       IF #Sts_PosAxis = 2 AND NOT #Alarm.CheckBothAxMove THEN
               //
               #Ax_Testa.CIn.Manager.MoveToPos := #Ctrl.Ax.OP_MoveToPos AND #Sts.Op_MoveToPos_Cnd;
               #Ax_Coda.CIn.Manager.MoveToPos := #Ctrl.Ax.OP_MoveToPos AND #Sts.Op_MoveToPos_Cnd;
               #Ax_Testa.CIn.Manager.Pos := #Ax_Coda.CIn.Manager.Pos := #CIn.Manager.Pos;

       END_IF;


       // ##########################
   (*    
   IF #Ctrl.Ax.OP_MoveToPos AND #Sts.Op_MoveToPos_Cnd AND NOT #Ax_Testa.COut.InPosition AND #Sollevatore_Testa.COut.Rest
       AND ( NOT #Alarm.Testa.Ax.S120_Fault AND NOT #Alarm.Coda.Ax.S120_Fault) THEN
       #Ax_Testa.CIn.Manager.MoveToPos := TRUE;

       // Se raggiungo la posizione di setpoint spengo il comando
   ELSIF #Ax_Testa.COut.InPosition AND #Ax_Testa.COut.Standstill OR ( #Alarm.Testa.Ax.S120_Fault OR #Alarm.Coda.Ax.S120_Fault) THEN
       #Ax_Testa.CIn.Manager.MoveToPos := FALSE;
       #Ax_Testa.DSI.PowerEnable := FALSE;
   END_IF;

   // MANIPOLATORE CODA
   #Ax_Coda.CIn.Manager.Control_ON := #Ax_Coda.DSI.PowerEnable
   := #Sollevatore_Coda.Cin.Manager.Control_ON := #Magnete_Coda.Cin.Manager.Control_ON := #Ctrl.Ax.OP_MoveToPos;

   IF #Ctrl.Ax.OP_MoveToPos AND #Sts.Op_MoveToPos_Cnd AND NOT #Ax_Coda.COut.InPosition AND #Sollevatore_Coda.COut.Rest
       AND ( NOT #Alarm.Testa.Ax.S120_Fault AND NOT #Alarm.Coda.Ax.S120_Fault) THEN
           #Ax_Coda.CIn.Manager.MoveToPos := TRUE;

           // Se raggiungo la posizione di setpoint spengo il comando
       ELSIF #Ax_Coda.COut.InPosition AND #Ax_Coda.COut.Standstill OR ( #Alarm.Testa.Ax.S120_Fault OR #Alarm.Coda.Ax.S120_Fault) THEN
           #Ax_Coda.CIn.Manager.MoveToPos := FALSE;
           #Ax_Coda.DSI.PowerEnable := FALSE;
       END_IF;
       *)
END_REGION

REGION Network 55 (SCL): [Sollevamento] - Cin Manager (Esecuzione sequenza comandi)
   // Comando CIn Manager ControlON di tutte le utenze
   // MANIPOLATORE TESTA & CODA
   #Sollevatore_Testa.Cin.Manager.Control_ON := #CIn.Manager.Control_ON;
   #Sollevatore_Coda.Cin.Manager.Control_ON := #CIn.Manager.Control_ON;
   //
   #Sollevatore_Testa.Cin.Manager.Rest := FALSE;
   #Sollevatore_Testa.Cin.Manager.Work := FALSE;
   #Sollevatore_Coda.Cin.Manager.Rest := FALSE;
   #Sollevatore_Coda.Cin.Manager.Work := FALSE;

   // Gestione dei comandi relativi a Sollevamento in sequenza quando ho un OP cnd

   IF (#Ctrl.Sollevamento.OP_Rest AND #Sts.Sollevamento.OP_Rest_Cnd) THEN

       #Sollevatore_Testa.Cin.Manager.Rest := TRUE;
       #Sollevatore_Coda.Cin.Manager.Rest := TRUE;

           // Vado a lavoro solo se sono in posizione    
   ELSIF  (#Ctrl.Sollevamento.OP_Work AND #Sts.Sollevamento.Op_Work_Cnd) AND (#COut.InPos_Prelievo OR #COut.InPos_BancoScarto OR #COut.InPos_BancoA0303) THEN

       #Sollevatore_Testa.Cin.Manager.Work := TRUE;
       #Sollevatore_Coda.Cin.Manager.Work := TRUE;

   END_IF;
END_REGION

REGION Network 56 (SCL): [Magneti] - Cin Manager (Esecuzione sequenza comandi)


   // Comando CIn Manager ControlON di tutte le utenze
   // MAGNETI TESTA & CODA
   #Magnete_Testa.Cin.Manager.Control_ON := (#Ctrl.Magneti.OP_Rest OR #Ctrl.Magneti.OP_Work) OR (#Ctrl.Sollevamento.OP_Rest OR #Ctrl.Sollevamento.OP_Work);
   #Magnete_Coda.Cin.Manager.Control_ON := (#Ctrl.Magneti.OP_Rest OR #Ctrl.Magneti.OP_Work) OR (#Ctrl.Sollevamento.OP_Rest OR #Ctrl.Sollevamento.OP_Work);
   //
   // Gestione dei comandi relativi ai Magneti in sequenza quando ho un OP cnd
   IF (#Ctrl.Magneti.OP_Rest AND #Sts.Magneti.OP_Rest_Cnd) AND #Sollevatore_Testa.COut.Work AND #Sollevatore_Coda.COut.Work THEN

       #Magnete_Testa.Cin.Manager.Work := FALSE;
       #Magnete_Coda.Cin.Manager.Work := FALSE;
       #Magnete_Testa.Cin.Manager.Rest := TRUE;
       #Magnete_Coda.Cin.Manager.Rest := TRUE;

   ELSIF (#Ctrl.Magneti.OP_Rest AND #Sts.Magneti.OP_Rest_Cnd) AND #COut.InPos_BancoScarto THEN

       #Magnete_Testa.Cin.Manager.Work := FALSE;
       #Magnete_Coda.Cin.Manager.Work := FALSE;
       #Magnete_Testa.Cin.Manager.Rest := TRUE;
       #Magnete_Coda.Cin.Manager.Rest := TRUE;

           // Vado a lavoro solo se sono in posizione e il sollevatore è a lavoro    
   ELSIF  (#Ctrl.Magneti.OP_Work AND #Sts.Magneti.Op_Work_Cnd) THEN

       #Magnete_Testa.Cin.Manager.Rest := FALSE;
       #Magnete_Coda.Cin.Manager.Rest := FALSE;
       #Magnete_Testa.Cin.Manager.Work := TRUE;
       #Magnete_Coda.Cin.Manager.Work := TRUE;

   END_IF;
END_REGION

REGION Network 58: <<< MACHINE STATUS >>>
END_REGION

REGION Network 59: Collect machine to zone interface (internal machines OR)
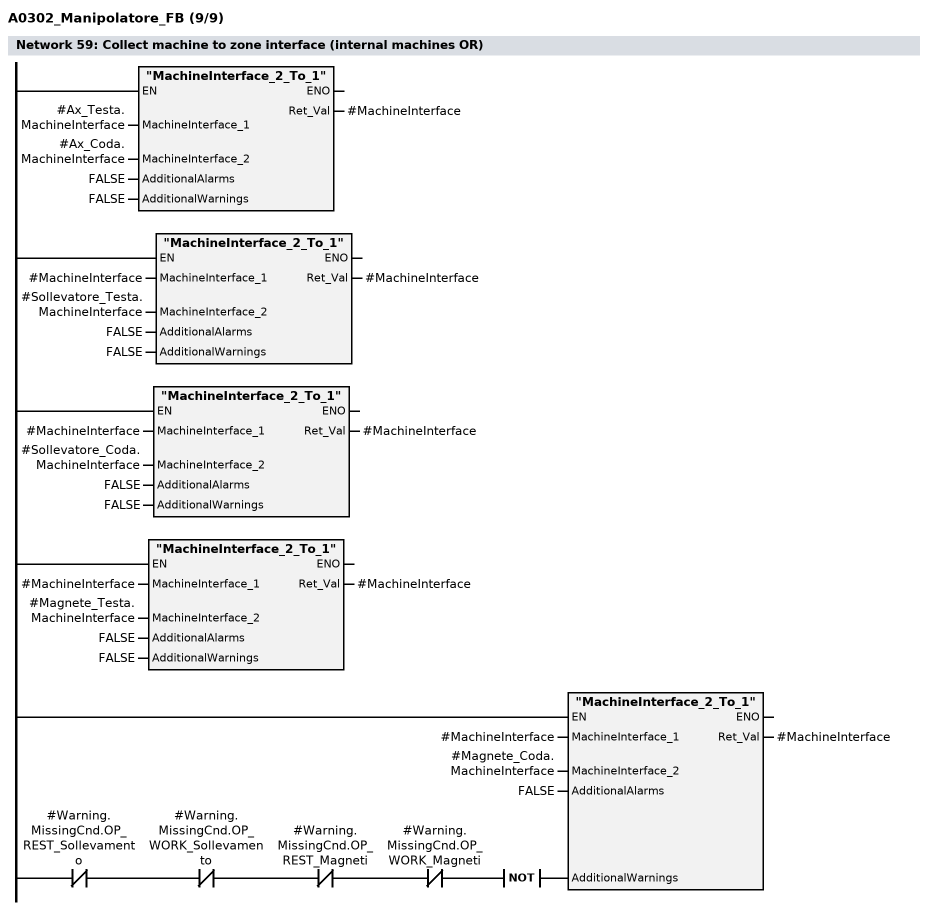
   RUNG wire#powerrail
      "MachineInterface_2_To_1"(MachineInterface_1 := #Ax_Testa.MachineInterface, MachineInterface_2 := #Ax_Coda.MachineInterface, AdditionalAlarms := FALSE, AdditionalWarnings := FALSE, Ret_Val => #MachineInterface)
   END_RUNG
   RUNG wire#powerrail
      "MachineInterface_2_To_1"(MachineInterface_1 := #MachineInterface, MachineInterface_2 := #Sollevatore_Testa.MachineInterface, AdditionalAlarms := FALSE, AdditionalWarnings := FALSE, Ret_Val => #MachineInterface)
   END_RUNG
   RUNG wire#powerrail
      "MachineInterface_2_To_1"(MachineInterface_1 := #MachineInterface, MachineInterface_2 := #Sollevatore_Coda.MachineInterface, AdditionalAlarms := FALSE, AdditionalWarnings := FALSE, Ret_Val => #MachineInterface)
   END_RUNG
   RUNG wire#powerrail
      "MachineInterface_2_To_1"(MachineInterface_1 := #MachineInterface, MachineInterface_2 := #Magnete_Testa.MachineInterface, AdditionalAlarms := FALSE, AdditionalWarnings := FALSE, Ret_Val => #MachineInterface)
   END_RUNG
   RUNG wire#powerrail
      "MachineInterface_2_To_1"(AdditionalWarnings := wire#w1, MachineInterface_1 := #MachineInterface, MachineInterface_2 := #Magnete_Coda.MachineInterface, AdditionalAlarms := FALSE, Ret_Val => #MachineInterface)
   END_RUNG
   RUNG wire#powerrail
      I_Contact( #Warning.MissingCnd.OP_REST_Sollevamento )
      I_Contact( #Warning.MissingCnd.OP_WORK_Sollevamento )
      I_Contact( #Warning.MissingCnd.OP_REST_Magneti )
      I_Contact( #Warning.MissingCnd.OP_WORK_Magneti )
      Not()
   END_RUNG wire#w1
   // the same network as SCL:
   #MachineInterface := "MachineInterface_2_To_1"(MachineInterface_1 := #Ax_Testa.MachineInterface,
                           MachineInterface_2 := #Ax_Coda.MachineInterface,
                           AdditionalAlarms := FALSE,
                           AdditionalWarnings := FALSE);
   #MachineInterface := "MachineInterface_2_To_1"(MachineInterface_1 := #MachineInterface,
                           MachineInterface_2 := #Sollevatore_Testa.MachineInterface,
                           AdditionalAlarms := FALSE,
                           AdditionalWarnings := FALSE);
   #MachineInterface := "MachineInterface_2_To_1"(MachineInterface_1 := #MachineInterface,
                           MachineInterface_2 := #Sollevatore_Coda.MachineInterface,
                           AdditionalAlarms := FALSE,
                           AdditionalWarnings := FALSE);
   #MachineInterface := "MachineInterface_2_To_1"(MachineInterface_1 := #MachineInterface,
                           MachineInterface_2 := #Magnete_Testa.MachineInterface,
                           AdditionalAlarms := FALSE,
                           AdditionalWarnings := FALSE);
   #MachineInterface := "MachineInterface_2_To_1"(MachineInterface_1 := #MachineInterface,
                           MachineInterface_2 := #Magnete_Coda.MachineInterface,
                           AdditionalAlarms := FALSE,
                           AdditionalWarnings := NOT (NOT #Warning.MissingCnd.OP_REST_Sollevamento AND NOT #Warning.MissingCnd.OP_WORK_Sollevamento AND NOT #Warning.MissingCnd.OP_REST_Magneti AND NOT #Warning.MissingCnd.OP_WORK_Magneti));
END_REGION
END_FUNCTION_BLOCK

FUNCTION "A0302_Bordatrice_RegolazioneFormato_OB1_CALL" : Void   // FC151, LAD
// stored: SetENOAutomatically false
   VAR_TEMP
      RETVAL_SET_CINT : Int;
      Check_Low : Bool;
      ChecK_High : Bool;
   END_VAR
   VAR_TEMP   // added for the SCL form of the ladder/FBD networks
      _w1 : Bool;
      _w2 : Bool;
      _w3 : Bool;
   END_VAR
BEGIN

REGION Network 2
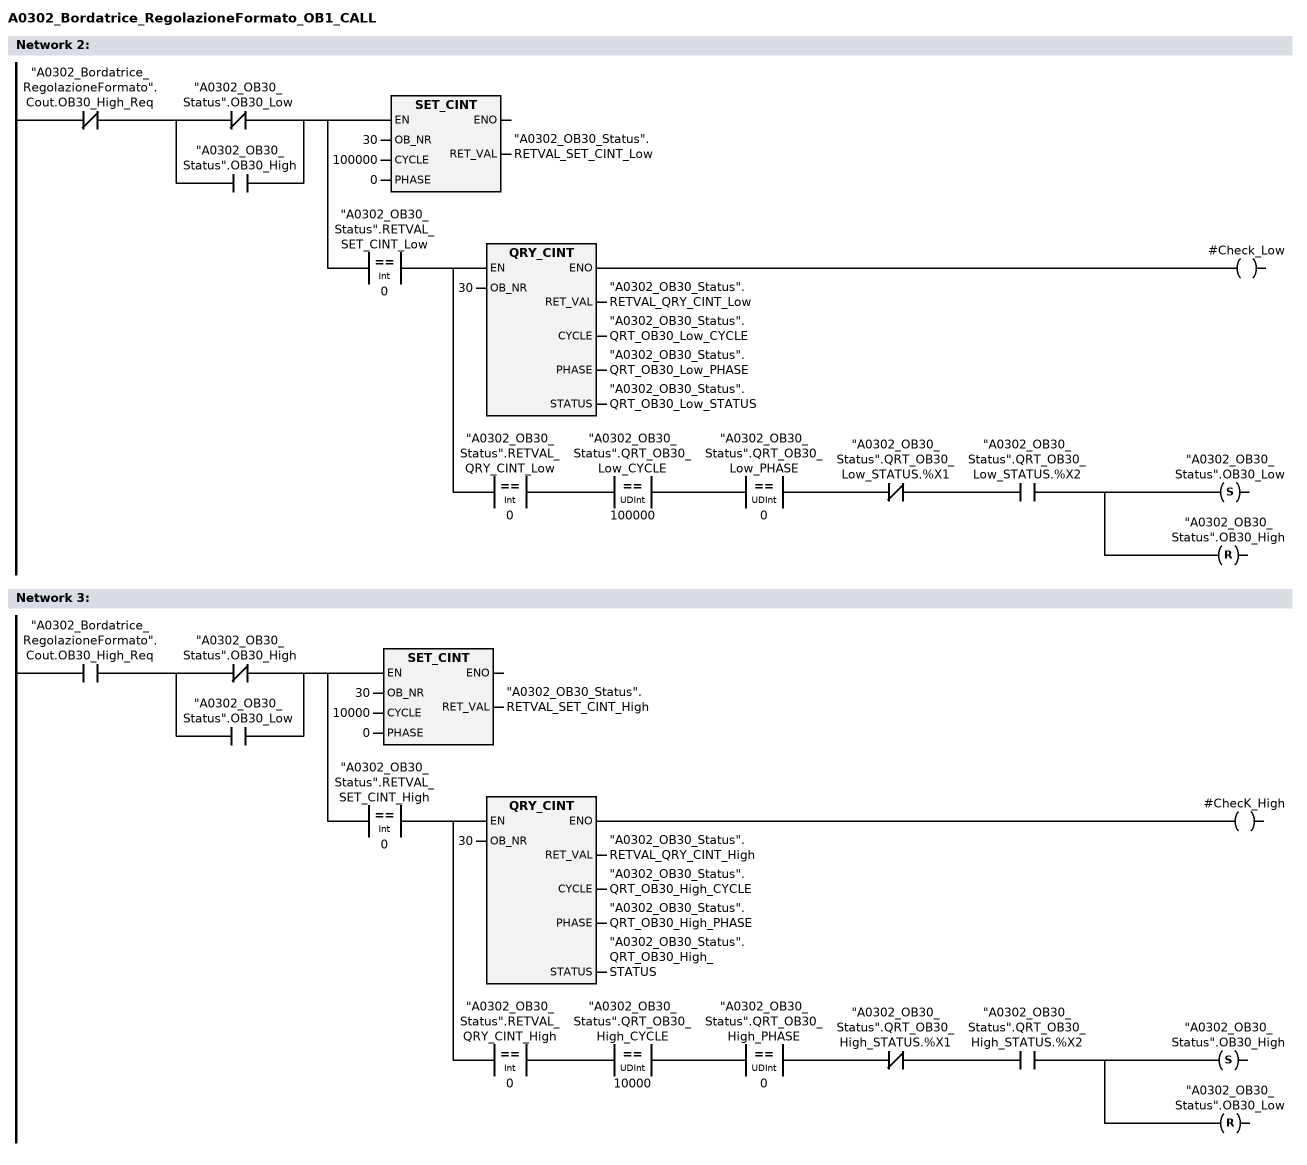
   RUNG wire#powerrail
      I_Contact( "A0302_Bordatrice_RegolazioneFormato".Cout.OB30_High_Req )
      wire#w1
      I_Contact( "A0302_OB30_Status".OB30_Low )
      wire#w2
      SET_CINT(OB_NR := 30, CYCLE := 100000, PHASE := 0, RET_VAL => "A0302_OB30_Status".RETVAL_SET_CINT_Low)
   END_RUNG
   RUNG wire#w1
      Contact( "A0302_OB30_Status".OB30_High )
   END_RUNG wire#w2
   RUNG wire#w2
      { S7_Templates := "SrcType := Int" } EQ_Contact(in1 := "A0302_OB30_Status".RETVAL_SET_CINT_Low, in2 := 0)
      wire#w3
      QRY_CINT(OB_NR := 30, RET_VAL => "A0302_OB30_Status".RETVAL_QRY_CINT_Low, CYCLE => "A0302_OB30_Status".QRT_OB30_Low_CYCLE, PHASE => "A0302_OB30_Status".QRT_OB30_Low_PHASE, STATUS => "A0302_OB30_Status".QRT_OB30_Low_STATUS)
      Coil( #Check_Low )
   END_RUNG
   RUNG wire#w3
      { S7_Templates := "SrcType := Int" } EQ_Contact(in1 := "A0302_OB30_Status".RETVAL_QRY_CINT_Low, in2 := 0)
      { S7_Templates := "SrcType := UDInt" } EQ_Contact(in1 := "A0302_OB30_Status".QRT_OB30_Low_CYCLE, in2 := 100000)
      { S7_Templates := "SrcType := UDInt" } EQ_Contact(in1 := "A0302_OB30_Status".QRT_OB30_Low_PHASE, in2 := 0)
      I_Contact( "A0302_OB30_Status".QRT_OB30_Low_STATUS.%X1 )
      Contact( "A0302_OB30_Status".QRT_OB30_Low_STATUS.%X2 )
      wire#w4
      S_Coil( "A0302_OB30_Status".OB30_Low )
   END_RUNG
   RUNG wire#w4
      R_Coil( "A0302_OB30_Status".OB30_High )
   END_RUNG
   // the same network as SCL:
   #_w1 := NOT "A0302_Bordatrice_RegolazioneFormato".Cout.OB30_High_Req AND (NOT "A0302_OB30_Status".OB30_Low OR "A0302_OB30_Status".OB30_High);
   IF #_w1 THEN
       "A0302_OB30_Status".RETVAL_SET_CINT_Low := SET_CINT(OB_NR := 30, CYCLE := 100000, PHASE := 0);
   END_IF;
   #_w2 := #_w1 AND ("A0302_OB30_Status".RETVAL_SET_CINT_Low = 0);
   "A0302_OB30_Status".RETVAL_QRY_CINT_Low := QRY_CINT(EN := #_w2,
                           OB_NR := 30,
                           CYCLE => "A0302_OB30_Status".QRT_OB30_Low_CYCLE,
                           PHASE => "A0302_OB30_Status".QRT_OB30_Low_PHASE,
                           STATUS => "A0302_OB30_Status".QRT_OB30_Low_STATUS,
                           ENO => #_w3);
   #Check_Low := #_w3;
   IF #_w2 AND ("A0302_OB30_Status".RETVAL_QRY_CINT_Low = 0) AND ("A0302_OB30_Status".QRT_OB30_Low_CYCLE = 100000) AND ("A0302_OB30_Status".QRT_OB30_Low_PHASE = 0) AND NOT "A0302_OB30_Status".QRT_OB30_Low_STATUS.%X1 AND "A0302_OB30_Status".QRT_OB30_Low_STATUS.%X2 THEN
       "A0302_OB30_Status".OB30_Low := TRUE;
       "A0302_OB30_Status".OB30_High := FALSE;
   END_IF;
END_REGION

REGION Network 3
   RUNG wire#powerrail
      Contact( "A0302_Bordatrice_RegolazioneFormato".Cout.OB30_High_Req )
      wire#w1
      I_Contact( "A0302_OB30_Status".OB30_High )
      wire#w2
      SET_CINT(OB_NR := 30, CYCLE := 10000, PHASE := 0, RET_VAL => "A0302_OB30_Status".RETVAL_SET_CINT_High)
   END_RUNG
   RUNG wire#w1
      Contact( "A0302_OB30_Status".OB30_Low )
   END_RUNG wire#w2
   RUNG wire#w2
      { S7_Templates := "SrcType := Int" } EQ_Contact(in1 := "A0302_OB30_Status".RETVAL_SET_CINT_High, in2 := 0)
      wire#w3
      QRY_CINT(OB_NR := 30, RET_VAL => "A0302_OB30_Status".RETVAL_QRY_CINT_High, CYCLE => "A0302_OB30_Status".QRT_OB30_High_CYCLE, PHASE => "A0302_OB30_Status".QRT_OB30_High_PHASE, STATUS => "A0302_OB30_Status".QRT_OB30_High_STATUS)
      Coil( #ChecK_High )
   END_RUNG
   RUNG wire#w3
      { S7_Templates := "SrcType := Int" } EQ_Contact(in1 := "A0302_OB30_Status".RETVAL_QRY_CINT_High, in2 := 0)
      { S7_Templates := "SrcType := UDInt" } EQ_Contact(in1 := "A0302_OB30_Status".QRT_OB30_High_CYCLE, in2 := 10000)
      { S7_Templates := "SrcType := UDInt" } EQ_Contact(in1 := "A0302_OB30_Status".QRT_OB30_High_PHASE, in2 := 0)
      I_Contact( "A0302_OB30_Status".QRT_OB30_High_STATUS.%X1 )
      Contact( "A0302_OB30_Status".QRT_OB30_High_STATUS.%X2 )
      wire#w4
      S_Coil( "A0302_OB30_Status".OB30_High )
   END_RUNG
   RUNG wire#w4
      R_Coil( "A0302_OB30_Status".OB30_Low )
   END_RUNG
   // the same network as SCL:
   #_w1 := "A0302_Bordatrice_RegolazioneFormato".Cout.OB30_High_Req AND (NOT "A0302_OB30_Status".OB30_High OR "A0302_OB30_Status".OB30_Low);
   IF #_w1 THEN
       "A0302_OB30_Status".RETVAL_SET_CINT_High := SET_CINT(OB_NR := 30, CYCLE := 10000, PHASE := 0);
   END_IF;
   #_w2 := #_w1 AND ("A0302_OB30_Status".RETVAL_SET_CINT_High = 0);
   "A0302_OB30_Status".RETVAL_QRY_CINT_High := QRY_CINT(EN := #_w2,
                           OB_NR := 30,
                           CYCLE => "A0302_OB30_Status".QRT_OB30_High_CYCLE,
                           PHASE => "A0302_OB30_Status".QRT_OB30_High_PHASE,
                           STATUS => "A0302_OB30_Status".QRT_OB30_High_STATUS,
                           ENO => #_w3);
   #ChecK_High := #_w3;
   IF #_w2 AND ("A0302_OB30_Status".RETVAL_QRY_CINT_High = 0) AND ("A0302_OB30_Status".QRT_OB30_High_CYCLE = 10000) AND ("A0302_OB30_Status".QRT_OB30_High_PHASE = 0) AND NOT "A0302_OB30_Status".QRT_OB30_High_STATUS.%X1 AND "A0302_OB30_Status".QRT_OB30_High_STATUS.%X2 THEN
       "A0302_OB30_Status".OB30_High := TRUE;
       "A0302_OB30_Status".OB30_Low := FALSE;
   END_IF;
END_REGION
END_FUNCTION

FUNCTION "A0302_Bordatrice_CALL" : Void   // FC181, LAD
TITLE = << BORDATRICE MOVIMENTO >>
// stored: SetENOAutomatically false
   VAR CONSTANT
      MinimumPos : Real := 0.0;
      MaximumPos : Real := 1000.0;
      MISSING : Int;
   END_VAR
BEGIN

REGION Network 1 (SCL): << TRASFERIMENTO stati CIn del blocco >>
   // SOSTITUIRE SYS BYPASS CON INGRESSI DIGITALI

   // TRASFERIMENTO COMANDI CIn MANAGER
   "A0302_Bordatrice".CIn.Manager.Ax := "A0302_Manager".COut.Bordatrice.Ax;
   //
   "A0302_Bordatrice".CIn.SemiAut_Pb := "A0302_Manager".DataIn.SemiAut_Pb;


   REGION TRASFERIMENTO CIn DIGITAL INPUT dei LIMIT SWITCH
       //
       //"A0302_Bordatrice".Ax.CIn.PositionLimits.EnableMin := FALSE;
       //"A0302_Bordatrice".Ax.CIn.PositionLimits.EnableMax := FALSE;

   END_REGION ;

   REGION TRASFERIMENTO STATI STAZIONE P5

       "A0302_Bordatrice".CIn.P5.Sollevatori := "A0301_Spintore_Lat".COut.Sollevatori;
       "A0302_Bordatrice".CIn.P5.SpintoreLong := "A0302_Spintore".COut.Spintore;
       "A0302_Bordatrice".CIn.P5.Sens.FTC_Ingombro_A0301 := "A0302_Spintore".IEC.FTC_On;

   END_REGION ;

   REGION  TRASFERIMENTO STATI RULLIERA dopo BORDATRICE

       "A0302_Bordatrice".CIn.Rulliera.Centratori := "A0302_Centratori".COut.Centraggio;
       "A0302_Bordatrice".CIn.Rulliera.Sollevatori := "A0302_Centratori".COut.Sollevamento;
       "A0302_Bordatrice".CIn.Rulliera.Coda.Sens := "A0302_Manager".CIn.Rulliera.Coda.Sens;
       "A0302_Bordatrice".CIn.Rulliera.Centro.Sens := "A0302_Manager".CIn.Rulliera.Centro.Sens;

   END_REGION ;

   REGION TRASFERIMENTO STATI CARRO PAREGGIATORE DI CODA

       "A0302_Bordatrice".CIn.CarroPareggCoda.Ax := "A0302_PareggiatoreCoda".COut.Ax;
       "A0302_Bordatrice".CIn.CarroPareggCoda.Bloccaggio := "A0302_PareggiatoreCoda".COut.Bloccaggio;
       "A0302_Bordatrice".CIn.CarroPareggCoda.BattutaVerticale := "A0302_PareggiatoreCoda".COut.BattutaVerticale;
       "A0302_Bordatrice".CIn.CarroPareggCoda.PareggiatoreLongitudinale := "A0302_PareggiatoreCoda".COut.PareggiatoreLong;
       "A0302_Bordatrice".CIn.CarroPareggCoda.Sens := "A0302_Manager".CIn.CarroPareggCoda.Sens;

   END_REGION ;

   REGION  TRASFERIMENTO STATI CARRO PAREGGIATORE DI TESTA

       "A0302_Bordatrice".CIn.CarroPareggTesta.Ax := "A0302_PareggiatoreTesta".COut.Ax;
       "A0302_Bordatrice".CIn.CarroPareggTesta.Bloccaggio := "A0302_PareggiatoreTesta".COut.Bloccaggio;
       "A0302_Bordatrice".CIn.CarroPareggTesta.Centraggio := "A0302_PareggiatoreTesta".COut.Centraggio;
       "A0302_Bordatrice".CIn.CarroPareggTesta.Sollevatore := "A0302_PareggiatoreTesta".COut.Sollevatore;
       "A0302_Bordatrice".CIn.CarroPareggTesta.Sens := "A0302_Manager".CIn.CarroPareggTesta.Sens;

   END_REGION ;

   // ATTREZZAGGIO PRONTO
   "A0302_Bordatrice".CIn.Attrezzaggio.CarriParegg.Ready := "A0302_Manager".Sts.Attrezzamento.Ready;
END_REGION

REGION Network 2 (SCL): << TRASFERIMENTO stati DataIn >>
   REGION TRASFERIMENTO #DataIn STATI BUTTON BORDATRICE
       // PB BORDATRICE
       "A0302_Bordatrice".Ax.DataIn.PB.Bwd_Minus := "A03_HMI".MB3.Button.A0302.Bordatrice.Ax.Bwd_Minus;
       "A0302_Bordatrice".Ax.DataIn.PB.Fwd_Plus := "A03_HMI".MB3.Button.A0302.Bordatrice.Ax.Fwd_Plus;
       "A0302_Bordatrice".Ax.DataIn.PB.MoveToPos := "A03_HMI".MB3.Button.A0302.Bordatrice.Ax.MoveToPos;

       // Sensori
       "A0302_Bordatrice".DataIn.Sens.FTC_Uscita := "A0302_Bordatrice_Banco_4_Lato_1_Phc_AtExit";

       // Feedback connettori
       "A0302_Bordatrice".DataIn.FdBack.ConnMotori := "A0302_Bordatrice_ControlloConnettoreBanco_4_Lato_1";
       "A0302_Bordatrice".DataIn.FdBack.ConnAux := "A0302_Bordatrice_ControlloConnettoreBanco_4_Lato_2";

   END_REGION ;
END_REGION

REGION Network 3 (SCL): DSI
   //
   "A0302_Bordatrice".DSI := "F_DB".DSI_S120_Bordatrice;
END_REGION

REGION Network 4 (SCL): HW
   //
   "A0302_Bordatrice".HWID_TEL111 := "HW_Const_Values".CU5_PN_1950A1_SIEMENS_telegram_111;
END_REGION

REGION Network 5 (SCL): Drive
   //
   "A0302_Bordatrice".Drive.Infeed_ON := "Areas_ITF".AG.Infeed_Running;
   "A0302_Bordatrice".Drive.AccessPoint := "HW_Const_Values".CU5_PN_1950A1_ModuleAccessPoint;
   "A0302_Bordatrice".Drive.AxisID := "CU5_ID_2_1950A1_1950M1";
   "A0302_Bordatrice".Drive.TokenChain := "TOKENCHAIN_CU5";
END_REGION

REGION Network 6: [Bordatrice] - Machine call
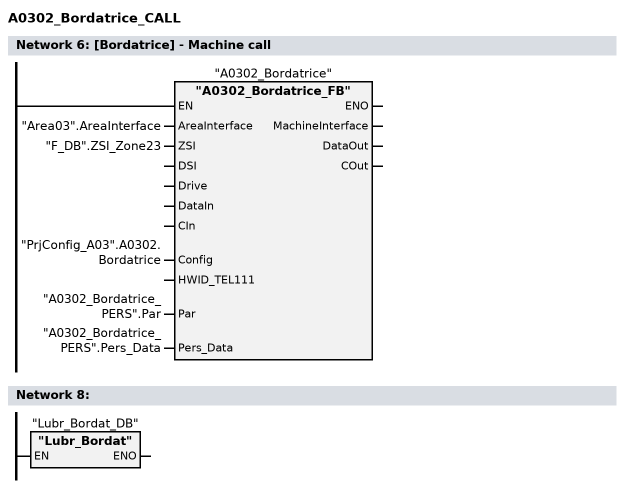
   RUNG wire#powerrail
      "A0302_Bordatrice"(AreaInterface := "Area03".AreaInterface, ZSI := "F_DB".ZSI_Zone23, DSI :=, Drive :=, DataIn :=, CIn :=, Config := "PrjConfig_A03".A0302.Bordatrice, HWID_TEL111 :=, Par := "A0302_Bordatrice_PERS".Par, Pers_Data := "A0302_Bordatrice_PERS".Pers_Data, MachineInterface =>, DataOut =>, COut =>)
   END_RUNG
   // the same network as SCL:
   "A0302_Bordatrice"(AreaInterface := "Area03".AreaInterface,   // "A0302_Bordatrice_FB"
                      ZSI := "F_DB".ZSI_Zone23,
                      Config := "PrjConfig_A03".A0302.Bordatrice,
                      Par := "A0302_Bordatrice_PERS".Par,
                      Pers_Data := "A0302_Bordatrice_PERS".Pers_Data);
END_REGION

REGION Network 8
   RUNG wire#powerrail
      "Lubr_Bordat_DB"()
   END_RUNG
   // the same network as SCL:
   "Lubr_Bordat_DB"();   // "Lubr_Bordat"
END_REGION
END_FUNCTION

FUNCTION_BLOCK "A0302_Bordatrice_FB"   // FB2, LAD
TITLE = == GESTIONE DELLA STAZIONE BORDATRICE ==
// stored: MemoryReserve 100, SetENOAutomatically false
   VAR_INPUT
      AreaInterface : "AreaInterface";
      ZSI : "udt_ZoneSafetyInterface";
      DSI : "udt_DeviceSafetyInterface";
      Drive : "TAx_DriveInterface";
      DataIn : Struct
         OP : "Ax_PB";
         Sens { ExternalAccessible := 'False'; ExternalVisible := 'False'; ExternalWritable := 'False'} : Struct
            FTC_Uscita : Bool;
         END_STRUCT;
         FdBack : Struct
            ConnMotori : Bool;
            ConnAux : Bool;
         END_STRUCT;
      END_STRUCT;
      CIn { ExternalAccessible := 'False'; ExternalVisible := 'False'; ExternalWritable := 'False'} : Struct
         Manager : Struct
            Ax : "Positioning_EPOS_Machine_Manager";
            Ax_Req : Struct
               Pos0 : Bool;
               Pos1 : Bool;
               Pos2 : Bool;
               Pos3 : Bool;
            END_STRUCT;
         END_STRUCT;
         SemiAut_Pb : Bool;
         P5 : Struct
            Sollevatori : "ValveMachine_COut";
            SpintoreLong : "ValveMachine_COut";
            Sens : Struct
               FTC_Ingombro_A0301 : Bool;   // 1614BF1 - I50.7
            END_STRUCT;
         END_STRUCT;
         Rulliera : Struct
            Ax_1 : "SpeedMachine_COut";
            Centratori : "ValveMachine_COut";
            Sollevatori : "ValveMachine_COut";
            Coda : Struct
               Sens : Struct
                  FTC_Rall : Bool;   // Sensori presenza materiale banco rallentamento ingresso
                  FTC_Prox_Ing : Bool;   // Sensori presenza materiale banco limite ingresso
               END_STRUCT;
            END_STRUCT;
            Centro : Struct
               Sens : Struct
                  FTC_Centrale : Bool;   // 2010BF1 - I50.2
               END_STRUCT;
            END_STRUCT;
         END_STRUCT;
         CarroPareggCoda : Struct
            Ax : "Positioning_DOL_Machine_COut";
            Bloccaggio : "ValveMachine_COut";
            BattutaVerticale : "ValveMachine_COut";
            PareggiatoreLongitudinale : "ValveMachine_COut";
            Sens : Struct
               FTC_Ingombro_In : Bool;   // 2012BF1 - I50.0
               FTC_Ingombro_Out : Bool;   // 2012BF2 - I50.1
               PresenzaMat : Bool;   // FC presenza materiale agganciato lato paregg coda
               PosPareggLong : Struct
                  Value : LReal;
                  CheckMeasure : Bool;
                  Standstill : Bool;
               END_STRUCT;
            END_STRUCT;
         END_STRUCT;
         CarroPareggTesta : Struct
            Ax : "Positioning_DOL_Machine_COut";
            Bloccaggio : "ValveMachine_COut";
            Centraggio : "ValveMachine_COut";
            Sollevatore : "ValveMachine_COut";
            Sens : Struct
               FTC1_Rall : Bool;   // 2010BF2 - I50.3
               FTC2_Prox_Ls : Bool;   // 2010BF3 - I50.4
               PresenzaMat : Bool;   // FC presenza materiale agganciato lato paregg testa
            END_STRUCT;
         END_STRUCT;
         Attrezzaggio : Struct
            CarriParegg : Struct
               Ready : Bool;
            END_STRUCT;
            BordRegFormato : Struct
               Ready : Bool;
            END_STRUCT;
         END_STRUCT;
      END_STRUCT;
      Config : Struct
         Ax : "Positioning_EPOS_Machine_Config_NEW";
         Measure : Struct
            K1_CarroPost : LReal;   // K1: Misura tra carro di coda e sensore applicato per controllo ingombro pezzo con carro giù
            K2_BancoIngresso : LReal;   // K2: Misura interasse tra lo 0 al centro del banco e la FTC all'uscita della Bordatrice
         END_STRUCT;
      END_STRUCT;
      HWID_TEL111 : HW_SUBMODULE;
   END_VAR
   VAR_OUTPUT
      MachineInterface { ExternalAccessible := 'False'; ExternalVisible := 'False'; ExternalWritable := 'False'} : "MachineInterface";
      DataOut : "Positioning_EPOS_Machine_DataOut";
      COut : Struct
         Ax : "Positioning_EPOS_Machine_COut";
         Ax_VelOveride : Struct
            Enable : Bool;
            Value : Real;
         END_STRUCT;
         Sts : Struct
            PosTargetEnable : Bool;
            PosTarget_Reached : Bool;
            In_W_Pos : Bool;
            AtRest : Bool;
         END_STRUCT;
         DataOut : "Positioning_EPOS_Machine_DataOut";
      END_STRUCT;
   END_VAR
   VAR_IN_OUT
      Par : Struct
         Ax_Man : "Positioning_EPOS_Machine_Par";
         Ax_Aut : "A0301_Mach_Speed_Par";
      END_STRUCT;
      Pers_Data : Struct
         EncoderAbsolute_Preset_OK : Bool;
         Persistent_ActualPosition : LReal;
      END_STRUCT;
   END_VAR
   VAR
      Alarm : Struct
         Ax { ExternalVisible := 'False'} : "Positioning_EPOS_Machine_Alr";
         StopIngombroCarroCoda : Bool;
         ConnMotori_FdBack : Bool;
         ConnAux_FdBack : Bool;
      END_STRUCT;
      Warning : Struct
         Ax { S7_SetPoint := 'True'} : "Positioning_EPOS_Machine_Wng";
         OP_REST_MissingCnd : Bool;   // Mancanza comando arresto
         OP_WORK_MissingCnd : Bool;   // Mancanza consenso lavoro
      END_STRUCT;
      Ax { S7_SetPoint := 'True'} : "Positioning_EPOS_Machine_FB_NEW";
      ValueVelOvr { ExternalAccessible := 'False'; ExternalVisible := 'False'; ExternalWritable := 'False'} : Array[1..10] of Real;
      Sts : Struct
         ReadyForMove : Bool;   // Pronto al movimento
         OP_CanMoveFreely : Bool;
         OP_MoveToPos_Cnd : Bool;
         OP_Bwd_Cnd : Bool;
         OP_Fwd_Cnd : Bool;
         Pz_UscitaBord : Bool;   // Pezzo in uscita dalla Bordatrice
         StopBordatrice : Bool;   // Stop Bordatrice da controllo quota spazio rimanente su rulliera di coda
         StandbyBordatrice : Bool;
      END_STRUCT;
      Ctrl : Struct
         Bordatrice : Struct
            OP_Bwd_Man : Bool;
            OP_Fwd_Man : Bool;
            OP_Bwd_Aut : Bool;
            OP_Fwd_Aut : Bool;
            OP_Bwd_Run : Bool;
            OP_Fwd_Run : Bool;
            OP_MoveToPos : Bool;
         END_STRUCT;
         Value : Struct
            Ax_TargetLongPos { ExternalAccessible := 'False'; ExternalVisible := 'False'; ExternalWritable := 'False'} : LReal;
            QuotaInizioUscita : LReal;
            QuotaFineUscita : LReal;
            PosTarget : LReal;
            QuotaRimanenteRullieraCoda : LReal;
         END_STRUCT;
         PosTargetEnable : Bool;
      END_STRUCT;
      HMI : Struct
         Pos : LReal;
      END_STRUCT;
      AUX : Struct
         Bordatrice : Struct
            OP_Bwd_Minus_PB : Bool;
            OP_Fwd_Plus_PB : Bool;
            OP_MoveToPos_PB { ExternalAccessible := 'False'; ExternalVisible := 'False'; ExternalWritable := 'False'} : Bool;
         END_STRUCT;
         Measure : Struct
            QuotaInizio : Bool;
            QuotaFine : Bool;
         END_STRUCT;
      END_STRUCT;
      IEC_FTC_UscitaBordatrice : Struct
         TON_Delay : IEC_TIMER;
         TOF_Delay { S7_SetPoint := 'True'} : IEC_TIMER;
         FTC_On { S7_SetPoint := 'True'} : Bool;
      END_STRUCT;
      IEC_StandbyBordatrice : IEC_TIMER;
      BTrk_Item : Struct
         BLean : Real;
         O_ID : DInt;
      END_STRUCT;
   END_VAR
   VAR_TEMP
      PE : Struct
         Bordatrice : Struct
            OP_Bwd_Minus_PB : Bool;
            OP_Fwd_Plus_PB : Bool;
            OP_MoveToPos_PB : Bool;
         END_STRUCT;
      END_STRUCT;
      VelOvr_Max : Real;   // Velocità max trovata
      i : Int;
      j : Int;
      CostB : LReal;
      Module : LReal;
      M_PosAPlusCostB : LReal;
      BTrk_GetData : Struct
         indx : Int;   // Se trovato tra i TODO / ENDING / OUT questo è l'indice dove sono stati prelevati i dati
         Sts : Int;   // 0 = Non Trovato; 0 = ACT; 1 = TODO; 2=ENDING; 3 = OUT
         Item : "Prod_Item_small";
      END_STRUCT;
      PositioningStop : Bool;
      NoTrk_Bordatrice : Bool;
   END_VAR
   VAR_TEMP   // added for the SCL form of the ladder/FBD networks
      _w1 : Bool;
      _w2 : Bool;
      _w3 : Bool;
      _w4 : Bool;
      _w5 : Bool;
      _w6 : Bool;
   END_VAR
BEGIN

REGION Network 1 (SCL): Reset allarmi
   IF #AreaInterface.RstAlarms THEN
       #Alarm.StopIngombroCarroCoda := FALSE;

       IF #DataIn.FdBack.ConnMotori AND #Alarm.ConnMotori_FdBack THEN
           #Alarm.ConnMotori_FdBack := FALSE;
       END_IF;

       IF #DataIn.FdBack.ConnAux AND #Alarm.ConnAux_FdBack THEN
           #Alarm.ConnAux_FdBack := FALSE;
       END_IF;
   END_IF;
   //
END_REGION

REGION Network 2: Controllo FdBack connettori
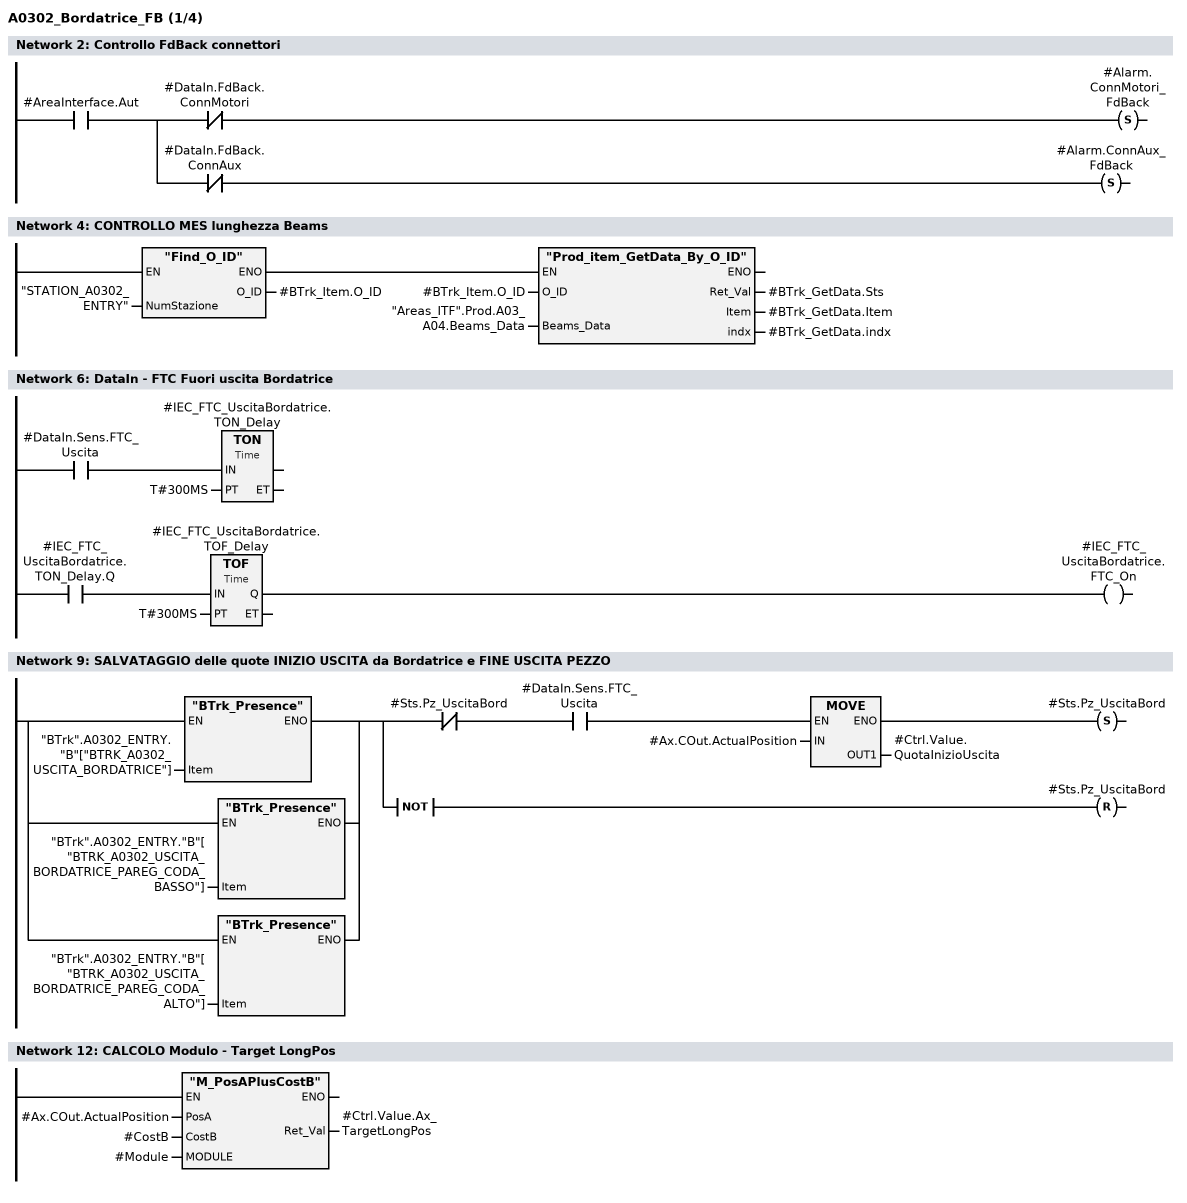
   RUNG wire#powerrail
      Contact( #AreaInterface.Aut )
      wire#w1
      I_Contact( #DataIn.FdBack.ConnMotori )
      S_Coil( #Alarm.ConnMotori_FdBack )
   END_RUNG
   RUNG wire#w1
      I_Contact( #DataIn.FdBack.ConnAux )
      S_Coil( #Alarm.ConnAux_FdBack )
   END_RUNG
   // the same network as SCL:
   IF #AreaInterface.Aut AND NOT #DataIn.FdBack.ConnMotori THEN #Alarm.ConnMotori_FdBack := TRUE; END_IF;
   IF #AreaInterface.Aut AND NOT #DataIn.FdBack.ConnAux THEN #Alarm.ConnAux_FdBack := TRUE; END_IF;
END_REGION

REGION Network 3: <+>
END_REGION

REGION Network 4: CONTROLLO MES lunghezza Beams
   RUNG wire#powerrail
      "Find_O_ID"(NumStazione := "STATION_A0302_ENTRY", O_ID => #BTrk_Item.O_ID)
      "Prod_item_GetData_By_O_ID"(O_ID := #BTrk_Item.O_ID, Beams_Data := "Areas_ITF".Prod.A03_A04.Beams_Data, Ret_Val => #BTrk_GetData.Sts, Item => #BTrk_GetData.Item, indx => #BTrk_GetData.indx)
   END_RUNG
   // the same network as SCL:
   "Find_O_ID"(NumStazione := "STATION_A0302_ENTRY", O_ID => #BTrk_Item.O_ID, ENO => #_w1);
   IF #_w1 THEN
       #BTrk_GetData.Sts := "Prod_item_GetData_By_O_ID"(O_ID := #BTrk_Item.O_ID,
                               Beams_Data := "Areas_ITF".Prod.A03_A04.Beams_Data,
                               Item => #BTrk_GetData.Item,
                               indx => #BTrk_GetData.indx);
   END_IF;
END_REGION

REGION Network 5 (SCL): CONTROLLO TRK lunghezza Beams
   //
   FOR #j:= 1 TO "BTRK_A0302_ENTRY_ITEMS" DO
       // 
       IF "BTrk".A0302_ENTRY.B[#j].BLen_Meas <> 0 THEN
           #BTrk_Item.BLean := "BTrk".A0302_ENTRY.B[#j].BLen_Meas;
       END_IF;

   END_FOR;
END_REGION

REGION Network 6: DataIn - FTC Fuori uscita Bordatrice
   RUNG wire#powerrail
      Contact( #DataIn.Sens.FTC_Uscita )
      { S7_Templates := "time_type := Time" } #IEC_FTC_UscitaBordatrice.TON_Delay.TON(pt := T#300MS, et =>)
   END_RUNG
   RUNG wire#powerrail
      Contact( #IEC_FTC_UscitaBordatrice.TON_Delay.Q )
      { S7_Templates := "time_type := Time" } #IEC_FTC_UscitaBordatrice.TOF_Delay.TOF(pt := T#300MS, et =>)
      Coil( #IEC_FTC_UscitaBordatrice.FTC_On )
   END_RUNG
   // the same network as SCL:
   #IEC_FTC_UscitaBordatrice.TON_Delay.TON(IN := #DataIn.Sens.FTC_Uscita, PT := T#300MS);
   #IEC_FTC_UscitaBordatrice.TOF_Delay.TOF(IN := #IEC_FTC_UscitaBordatrice.TON_Delay.Q, PT := T#300MS);
   #IEC_FTC_UscitaBordatrice.FTC_On := #IEC_FTC_UscitaBordatrice.TOF_Delay.Q;
END_REGION

REGION Network 7: <<<< CALCOLI QUOTE >>>>
END_REGION

REGION Network 8: <+>
END_REGION

REGION Network 9: SALVATAGGIO delle quote INIZIO USCITA da Bordatrice e FINE USCITA PEZZO
   RUNG wire#powerrail
      "BTrk_Presence"(Item := "BTrk".A0302_ENTRY."B"["BTRK_A0302_USCITA_BORDATRICE"])
      wire#w1
      I_Contact( #Sts.Pz_UscitaBord )
      Contact( #DataIn.Sens.FTC_Uscita )
      Move(in := #Ax.COut.ActualPosition, out1 => #Ctrl.Value.QuotaInizioUscita)
      S_Coil( #Sts.Pz_UscitaBord )
   END_RUNG
   RUNG wire#powerrail
      "BTrk_Presence"(Item := "BTrk".A0302_ENTRY."B"["BTRK_A0302_USCITA_BORDATRICE_PAREG_CODA_BASSO"])
   END_RUNG wire#w1
   RUNG wire#powerrail
      "BTrk_Presence"(Item := "BTrk".A0302_ENTRY."B"["BTRK_A0302_USCITA_BORDATRICE_PAREG_CODA_ALTO"])
   END_RUNG wire#w1
   RUNG wire#w1
      Not()
      R_Coil( #Sts.Pz_UscitaBord )
   END_RUNG
   // the same network as SCL:
   "BTrk_Presence"(Item := "BTrk".A0302_ENTRY."B"["BTRK_A0302_USCITA_BORDATRICE"], ENO => #_w1);
   "BTrk_Presence"(Item := "BTrk".A0302_ENTRY."B"["BTRK_A0302_USCITA_BORDATRICE_PAREG_CODA_BASSO"], ENO => #_w2);
   "BTrk_Presence"(Item := "BTrk".A0302_ENTRY."B"["BTRK_A0302_USCITA_BORDATRICE_PAREG_CODA_ALTO"], ENO => #_w3);
   #_w4 := #_w1 OR #_w2 OR #_w3;
   IF #_w4 AND NOT #Sts.Pz_UscitaBord AND #DataIn.Sens.FTC_Uscita THEN
       #Ctrl.Value.QuotaInizioUscita := #Ax.COut.ActualPosition;
       #Sts.Pz_UscitaBord := TRUE;
   END_IF;
   IF NOT #_w4 THEN #Sts.Pz_UscitaBord := FALSE; END_IF;
END_REGION

REGION Network 10 (SCL): CALCOLO dello spazio rimanete rulliera di coda
   (*** Calcolo quota Target pezzo - Se ho il carro di coda basso il target è pari alla lunghezza del pezzo
   IF #Sts.Pz_UscitaBord THEN
       #Ctrl.Value.PosTarget := #Ctrl.Value.QuotaInizioUscita + #BTrk_Item.BLean;
    END_IF; ***)

   // Calcolo dello Spazio prima del Pareggiatore di coda quando è in posizione
   // 
   #Ctrl.Value.QuotaRimanenteRullieraCoda := ((#Config.Measure.K2_BancoIngresso - #Config.Measure.K1_CarroPost) - #CIn.CarroPareggCoda.Ax.ActualPosition - 200.0);
   //
END_REGION

REGION Network 11 (SCL): CALCOLO Posizioni Target per lavoro Bordatrice
   // ******************************************************************
   // Calcoli del modulo
   // 

   #Module := #Ax.Config.Ax.Modulo_S120_P2566 / 1000.0;
   #CostB := (#Module / 2) - 1000.0;

   // Calcolo quota Target pezzo
   // Se ho il carro di coda basso il target è pari alla lunghezza del pezzo
   // 
   IF #Sts.Pz_UscitaBord THEN

       IF #CIn.CarroPareggCoda.BattutaVerticale.Work OR NOT "A0302_Manager".Ctrl.TRK.BTrk.RulliereVode THEN

           #Ctrl.Value.PosTarget := "M_PosAPlusCostB"(PosA := #Ctrl.Value.QuotaInizioUscita, CostB := #Ctrl.Value.QuotaRimanenteRullieraCoda, MODULE := #Module);

           #COut.Sts.PosTargetEnable:=#Ctrl.PosTargetEnable := TRUE;

           // Se ho il carro di coda alto il target è superiore alla lunghezza del pezzo per arrivare in fondo alla rulliera
       ELSE

           #Ctrl.Value.PosTarget := #Ctrl.Value.Ax_TargetLongPos;
           #COut.Sts.PosTargetEnable := #Ctrl.PosTargetEnable := FALSE;

       END_IF;

   ELSE
       #Ctrl.Value.PosTarget := #Ctrl.Value.Ax_TargetLongPos;
       #COut.Sts.PosTargetEnable := #Ctrl.PosTargetEnable := FALSE;
   END_IF;
END_REGION

REGION Network 12: CALCOLO Modulo - Target LongPos
   RUNG wire#powerrail
      "M_PosAPlusCostB"(PosA := #Ax.COut.ActualPosition, CostB := #CostB, MODULE := #Module, Ret_Val => #Ctrl.Value.Ax_TargetLongPos)
   END_RUNG
   // the same network as SCL:
   #Ctrl.Value.Ax_TargetLongPos := "M_PosAPlusCostB"(PosA := #Ax.COut.ActualPosition,
                           CostB := #CostB,
                           MODULE := #Module);
END_REGION

REGION Network 13: <+>
END_REGION

REGION Network 14: [Ax] Sts - Standby Bordatrice per mancanza prodotto da lavorare
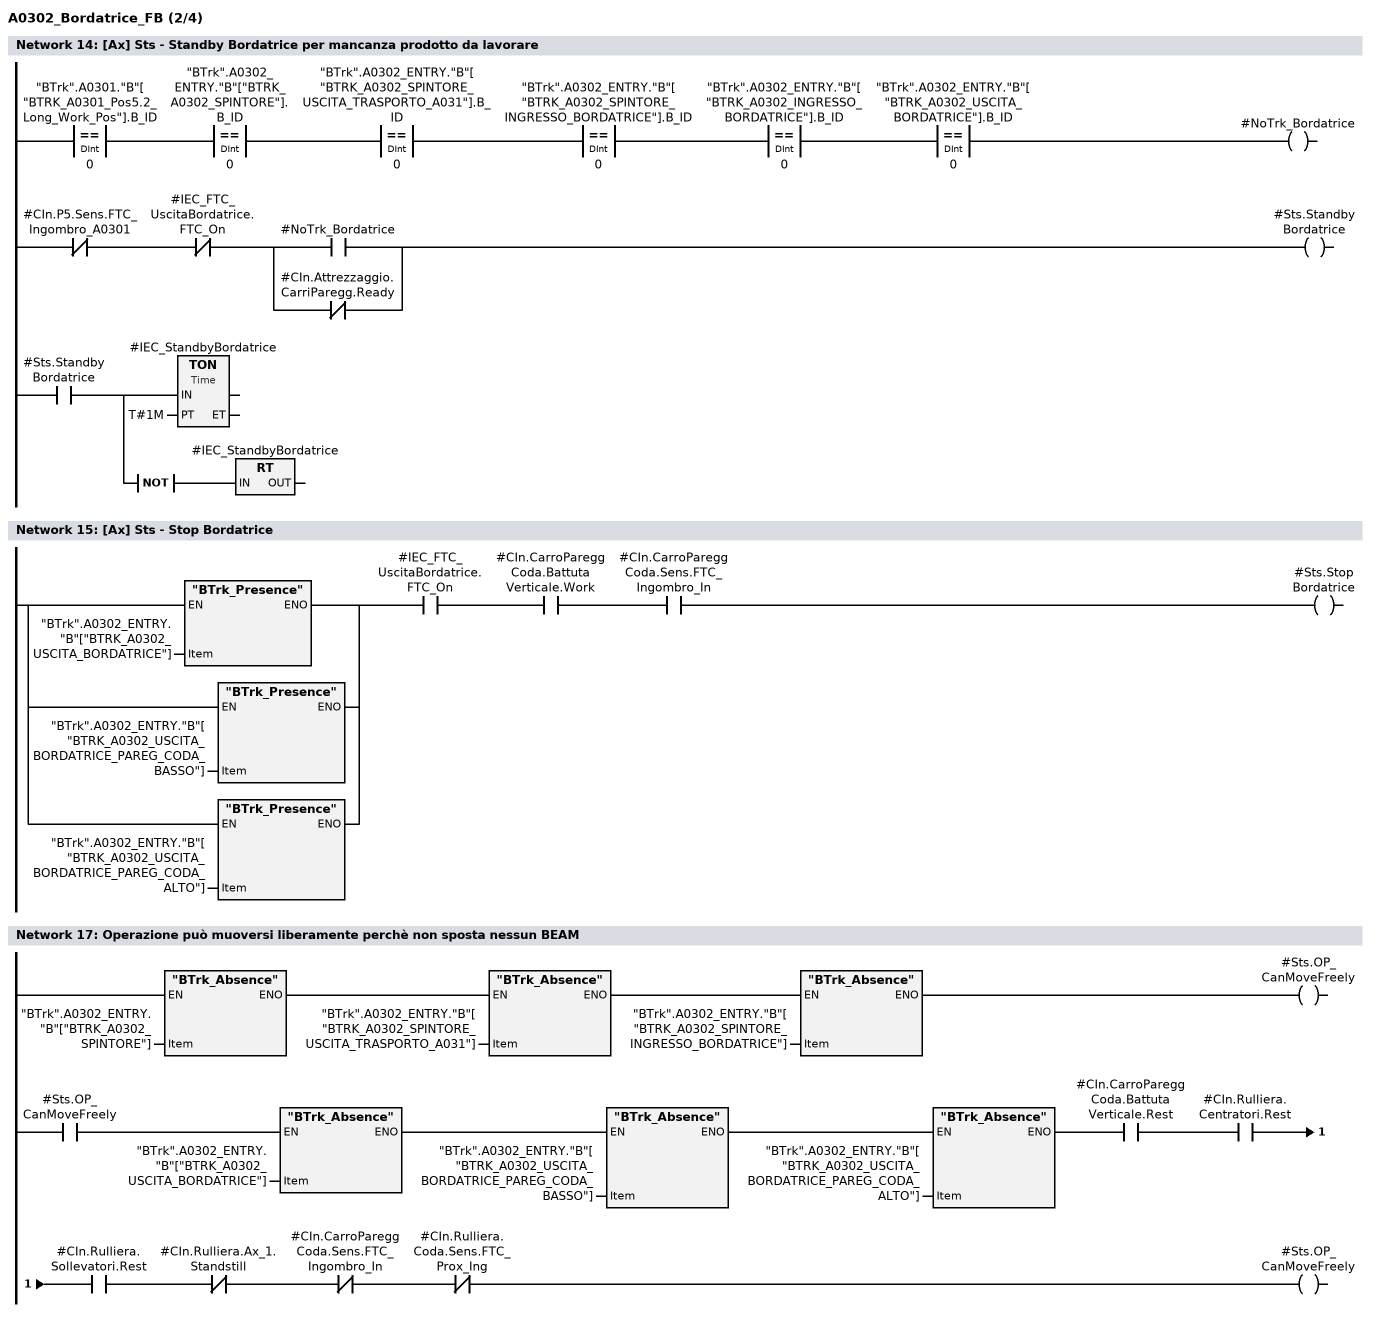
   RUNG wire#powerrail
      { S7_Templates := "SrcType := DInt" } EQ_Contact(in1 := "BTrk".A0301."B"["BTRK_A0301_Pos5.2_Long_Work_Pos"].B_ID, in2 := 0)
      { S7_Templates := "SrcType := DInt" } EQ_Contact(in1 := "BTrk".A0302_ENTRY."B"["BTRK_A0302_SPINTORE"].B_ID, in2 := 0)
      { S7_Templates := "SrcType := DInt" } EQ_Contact(in1 := "BTrk".A0302_ENTRY."B"["BTRK_A0302_SPINTORE_USCITA_TRASPORTO_A031"].B_ID, in2 := 0)
      { S7_Templates := "SrcType := DInt" } EQ_Contact(in1 := "BTrk".A0302_ENTRY."B"["BTRK_A0302_SPINTORE_INGRESSO_BORDATRICE"].B_ID, in2 := 0)
      { S7_Templates := "SrcType := DInt" } EQ_Contact(in1 := "BTrk".A0302_ENTRY."B"["BTRK_A0302_INGRESSO_BORDATRICE"].B_ID, in2 := 0)
      { S7_Templates := "SrcType := DInt" } EQ_Contact(in1 := "BTrk".A0302_ENTRY."B"["BTRK_A0302_USCITA_BORDATRICE"].B_ID, in2 := 0)
      Coil( #NoTrk_Bordatrice )
   END_RUNG
   RUNG wire#powerrail
      I_Contact( #CIn.P5.Sens.FTC_Ingombro_A0301 )
      I_Contact( #IEC_FTC_UscitaBordatrice.FTC_On )
      wire#w1
      Contact( #NoTrk_Bordatrice )
      wire#w2
      Coil( #Sts.StandbyBordatrice )
   END_RUNG
   RUNG wire#w1
      I_Contact( #CIn.Attrezzaggio.CarriParegg.Ready )
   END_RUNG wire#w2
   RUNG wire#powerrail
      Contact( #Sts.StandbyBordatrice )
      wire#w3
      { S7_Templates := "time_type := Time" } #IEC_StandbyBordatrice.TON(pt := T#1M, et =>)
   END_RUNG
   RUNG wire#w3
      Not()
      RT_Coil( #IEC_StandbyBordatrice )
   END_RUNG
   // the same network as SCL:
   #NoTrk_Bordatrice := ("BTrk".A0301."B"["BTRK_A0301_Pos5.2_Long_Work_Pos"].B_ID = 0) AND ("BTrk".A0302_ENTRY."B"["BTRK_A0302_SPINTORE"].B_ID = 0) AND ("BTrk".A0302_ENTRY."B"["BTRK_A0302_SPINTORE_USCITA_TRASPORTO_A031"].B_ID = 0) AND ("BTrk".A0302_ENTRY."B"["BTRK_A0302_SPINTORE_INGRESSO_BORDATRICE"].B_ID = 0) AND ("BTrk".A0302_ENTRY."B"["BTRK_A0302_INGRESSO_BORDATRICE"].B_ID = 0) AND ("BTrk".A0302_ENTRY."B"["BTRK_A0302_USCITA_BORDATRICE"].B_ID = 0);
   #Sts.StandbyBordatrice := NOT #CIn.P5.Sens.FTC_Ingombro_A0301 AND NOT #IEC_FTC_UscitaBordatrice.FTC_On AND (#NoTrk_Bordatrice OR NOT #CIn.Attrezzaggio.CarriParegg.Ready);
   #IEC_StandbyBordatrice.TON(IN := #Sts.StandbyBordatrice, PT := T#1M);
   IF NOT #Sts.StandbyBordatrice THEN RESET_TIMER(#IEC_StandbyBordatrice); END_IF;
END_REGION

REGION Network 15: [Ax] Sts - Stop Bordatrice
   RUNG wire#powerrail
      "BTrk_Presence"(Item := "BTrk".A0302_ENTRY."B"["BTRK_A0302_USCITA_BORDATRICE"])
      wire#w1
      Contact( #IEC_FTC_UscitaBordatrice.FTC_On )
      Contact( #CIn.CarroPareggCoda.BattutaVerticale.Work )
      Contact( #CIn.CarroPareggCoda.Sens.FTC_Ingombro_In )
      Coil( #Sts.StopBordatrice )
   END_RUNG
   RUNG wire#powerrail
      "BTrk_Presence"(Item := "BTrk".A0302_ENTRY."B"["BTRK_A0302_USCITA_BORDATRICE_PAREG_CODA_BASSO"])
   END_RUNG wire#w1
   RUNG wire#powerrail
      "BTrk_Presence"(Item := "BTrk".A0302_ENTRY."B"["BTRK_A0302_USCITA_BORDATRICE_PAREG_CODA_ALTO"])
   END_RUNG wire#w1
   // the same network as SCL:
   "BTrk_Presence"(Item := "BTrk".A0302_ENTRY."B"["BTRK_A0302_USCITA_BORDATRICE"], ENO => #_w1);
   "BTrk_Presence"(Item := "BTrk".A0302_ENTRY."B"["BTRK_A0302_USCITA_BORDATRICE_PAREG_CODA_BASSO"], ENO => #_w2);
   "BTrk_Presence"(Item := "BTrk".A0302_ENTRY."B"["BTRK_A0302_USCITA_BORDATRICE_PAREG_CODA_ALTO"], ENO => #_w3);
   #Sts.StopBordatrice := (#_w1 OR #_w2 OR #_w3) AND #IEC_FTC_UscitaBordatrice.FTC_On AND #CIn.CarroPareggCoda.BattutaVerticale.Work AND #CIn.CarroPareggCoda.Sens.FTC_Ingombro_In;
END_REGION

REGION Network 16: <+>
END_REGION

REGION Network 17: Operazione può muoversi liberamente perchè non sposta nessun BEAM
   RUNG wire#powerrail
      "BTrk_Absence"(Item := "BTrk".A0302_ENTRY."B"["BTRK_A0302_SPINTORE"])
      "BTrk_Absence"(Item := "BTrk".A0302_ENTRY."B"["BTRK_A0302_SPINTORE_USCITA_TRASPORTO_A031"])
      "BTrk_Absence"(Item := "BTrk".A0302_ENTRY."B"["BTRK_A0302_SPINTORE_INGRESSO_BORDATRICE"])
      Coil( #Sts.OP_CanMoveFreely )
   END_RUNG
   RUNG wire#powerrail
      Contact( #Sts.OP_CanMoveFreely )
      "BTrk_Absence"(Item := "BTrk".A0302_ENTRY."B"["BTRK_A0302_USCITA_BORDATRICE"])
      "BTrk_Absence"(Item := "BTrk".A0302_ENTRY."B"["BTRK_A0302_USCITA_BORDATRICE_PAREG_CODA_BASSO"])
      "BTrk_Absence"(Item := "BTrk".A0302_ENTRY."B"["BTRK_A0302_USCITA_BORDATRICE_PAREG_CODA_ALTO"])
      Contact( #CIn.CarroPareggCoda.BattutaVerticale.Rest )
      Contact( #CIn.Rulliera.Centratori.Rest )
      Contact( #CIn.Rulliera.Sollevatori.Rest )
      I_Contact( #CIn.Rulliera.Ax_1.Standstill )
      I_Contact( #CIn.CarroPareggCoda.Sens.FTC_Ingombro_In )
      I_Contact( #CIn.Rulliera.Coda.Sens.FTC_Prox_Ing )
      Coil( #Sts.OP_CanMoveFreely )
   END_RUNG
   // the same network as SCL:
   "BTrk_Absence"(Item := "BTrk".A0302_ENTRY."B"["BTRK_A0302_SPINTORE"], ENO => #_w1);
   "BTrk_Absence"(EN := #_w1,
                  Item := "BTrk".A0302_ENTRY."B"["BTRK_A0302_SPINTORE_USCITA_TRASPORTO_A031"],
                  ENO => #_w2);
   "BTrk_Absence"(EN := #_w2,
                  Item := "BTrk".A0302_ENTRY."B"["BTRK_A0302_SPINTORE_INGRESSO_BORDATRICE"],
                  ENO => #_w3);
   #Sts.OP_CanMoveFreely := #_w3;
   "BTrk_Absence"(EN := #Sts.OP_CanMoveFreely,
                  Item := "BTrk".A0302_ENTRY."B"["BTRK_A0302_USCITA_BORDATRICE"],
                  ENO => #_w4);
   "BTrk_Absence"(EN := #_w4,
                  Item := "BTrk".A0302_ENTRY."B"["BTRK_A0302_USCITA_BORDATRICE_PAREG_CODA_BASSO"],
                  ENO => #_w5);
   "BTrk_Absence"(EN := #_w5,
                  Item := "BTrk".A0302_ENTRY."B"["BTRK_A0302_USCITA_BORDATRICE_PAREG_CODA_ALTO"],
                  ENO => #_w6);
   #Sts.OP_CanMoveFreely := #_w6 AND #CIn.CarroPareggCoda.BattutaVerticale.Rest AND #CIn.Rulliera.Centratori.Rest AND #CIn.Rulliera.Sollevatori.Rest AND NOT #CIn.Rulliera.Ax_1.Standstill AND NOT #CIn.CarroPareggCoda.Sens.FTC_Ingombro_In AND NOT #CIn.Rulliera.Coda.Sens.FTC_Prox_Ing;
END_REGION

REGION Network 18: Comando Operazione Lavoro (AUT)
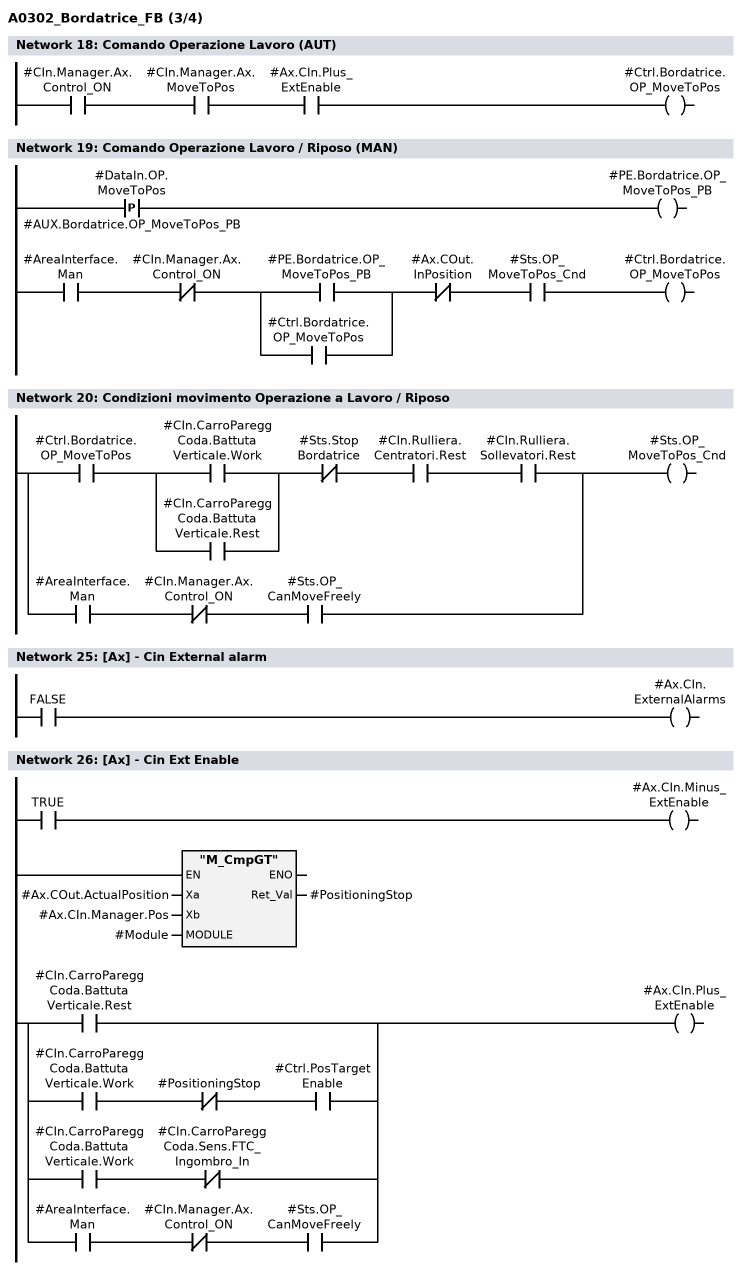
   RUNG wire#powerrail
      Contact( #CIn.Manager.Ax.Control_ON )
      Contact( #CIn.Manager.Ax.MoveToPos )
      Contact( #Ax.CIn.Plus_ExtEnable )
      Coil( #Ctrl.Bordatrice.OP_MoveToPos )
   END_RUNG
   // the same network as SCL:
   #Ctrl.Bordatrice.OP_MoveToPos := #CIn.Manager.Ax.Control_ON AND #CIn.Manager.Ax.MoveToPos AND #Ax.CIn.Plus_ExtEnable;
END_REGION

REGION Network 19: Comando Operazione Lavoro / Riposo (MAN)
   RUNG wire#powerrail
      P_Contact(operand := #DataIn.OP.MoveToPos, bit := #AUX.Bordatrice.OP_MoveToPos_PB)
      Coil( #PE.Bordatrice.OP_MoveToPos_PB )
   END_RUNG
   RUNG wire#powerrail
      Contact( #AreaInterface.Man )
      I_Contact( #CIn.Manager.Ax.Control_ON )
      wire#w1
      Contact( #PE.Bordatrice.OP_MoveToPos_PB )
      wire#w2
      I_Contact( #Ax.COut.InPosition )
      Contact( #Sts.OP_MoveToPos_Cnd )
      Coil( #Ctrl.Bordatrice.OP_MoveToPos )
   END_RUNG
   RUNG wire#w1
      Contact( #Ctrl.Bordatrice.OP_MoveToPos )
   END_RUNG wire#w2
   // the same network as SCL:
   #_w1 := #DataIn.OP.MoveToPos AND NOT #AUX.Bordatrice.OP_MoveToPos_PB;   // rising edge of #DataIn.OP.MoveToPos
   #AUX.Bordatrice.OP_MoveToPos_PB := #DataIn.OP.MoveToPos;
   #PE.Bordatrice.OP_MoveToPos_PB := #_w1;
   #Ctrl.Bordatrice.OP_MoveToPos := #AreaInterface.Man AND NOT #CIn.Manager.Ax.Control_ON AND (#PE.Bordatrice.OP_MoveToPos_PB OR #Ctrl.Bordatrice.OP_MoveToPos) AND NOT #Ax.COut.InPosition AND #Sts.OP_MoveToPos_Cnd;
END_REGION

REGION Network 20: Condizioni movimento Operazione a Lavoro / Riposo
   RUNG wire#powerrail
      Contact( #Ctrl.Bordatrice.OP_MoveToPos )
      wire#w1
      Contact( #CIn.CarroPareggCoda.BattutaVerticale.Work )
      wire#w2
      I_Contact( #Sts.StopBordatrice )
      Contact( #CIn.Rulliera.Centratori.Rest )
      Contact( #CIn.Rulliera.Sollevatori.Rest )
      wire#w3
      Coil( #Sts.OP_MoveToPos_Cnd )
   END_RUNG
   RUNG wire#w1
      Contact( #CIn.CarroPareggCoda.BattutaVerticale.Rest )
   END_RUNG wire#w2
   RUNG wire#powerrail
      Contact( #AreaInterface.Man )
      I_Contact( #CIn.Manager.Ax.Control_ON )
      Contact( #Sts.OP_CanMoveFreely )
   END_RUNG wire#w3
   // the same network as SCL:
   #Sts.OP_MoveToPos_Cnd := (#Ctrl.Bordatrice.OP_MoveToPos AND (#CIn.CarroPareggCoda.BattutaVerticale.Work OR #CIn.CarroPareggCoda.BattutaVerticale.Rest) AND NOT #Sts.StopBordatrice AND #CIn.Rulliera.Centratori.Rest AND #CIn.Rulliera.Sollevatori.Rest) OR (#AreaInterface.Man AND NOT #CIn.Manager.Ax.Control_ON AND #Sts.OP_CanMoveFreely);
END_REGION

REGION Network 21: <+>
END_REGION

REGION Network 22 (SCL): RIFERIMENTI [AX] - Positioning Manager
   // ******************************************************************************************
   REGION // TRASFERIMENTO DELLE RAMPE

       // Rampe in Manuale
       IF #AreaInterface.Man AND NOT #CIn.SemiAut_Pb THEN
           #Ax.Ctrl.Vel := #Par.Ax_Man.Man_Vel;
           #Ax.CIn.Manager.Acc := #Par.Ax_Man.Man_Acc;
           #Ax.CIn.Manager.Dec := #Par.Ax_Man.Man_Dec;
       END_IF;
   END_REGION

   // ******************************************************************************************
   REGION // // CALCOLO DELLA VELOCITA' TRASFERITA DALL'IMPIANTO IN BASE ALLA LUNGHEZZA DEL PEZZO

       // Inizializzo variabile di appoggio controllo overide massimo a un valore basso rispetto setpoint
       IF "Sys".AuxFirstPLCCycle THEN
           #VelOvr_Max := 100.0;
       END_IF;

       // Rallentamento Bordatrice con sensori
      (* 
       // Trasferisco velocità di rallentamento se ho posizionamento corto su pareggiatore di coda e raggiungo i sensori di rallentamento
       IF #Ax.#CIn.Manager.Control_ON AND #CIn.Manager.Ax.MoveToPos AND #CIn.CarroPareggCoda.BattutaVerticale.Work
           AND (#CIn.Rulliera.Coda.Sens.FTC_Rall OR #CIn.Rulliera.Coda.Sens.FTC_Prox_Ing) THEN
           #VelOvr_Max := 500.0;
       END_IF;

       // Trasferisco velocità di rallentamento se ho posizionamento lungo su pareggiatore di testa e raggiungo i sensori di rallentamento
       IF #CIn.Manager.Ax.MoveToPos AND #CIn.CarroPareggCoda.BattutaVerticale.Rest AND #CIn.Rulliera.Centro.Sens.FTC_Centrale
           AND (#CIn.CarroPareggTesta.Sens.FTC1_Rall OR #CIn.CarroPareggTesta.Sens.FTC2_Prox_Ls) THEN
           #VelOvr_Max := 500.0;
       END_IF;
       *)

       // Trasferisco le varibili su un array
       #ValueVelOvr[1] := "PPrf_MAIN".ON_WORK.A0301_A0302.Bordatrice.VelOvr_PLen_UpTo_1000;
       #ValueVelOvr[2] := "PPrf_MAIN".ON_WORK.A0301_A0302.Bordatrice.VelOvr_PLen_UpTo_1500;
       #ValueVelOvr[3] := "PPrf_MAIN".ON_WORK.A0301_A0302.Bordatrice.VelOvr_PLen_UpTo_2000;
       #ValueVelOvr[4] := "PPrf_MAIN".ON_WORK.A0301_A0302.Bordatrice.VelOvr_PLen_UpTo_2500;
       #ValueVelOvr[5] := "PPrf_MAIN".ON_WORK.A0301_A0302.Bordatrice.VelOvr_PLen_UpTo_3000;
       #ValueVelOvr[6] := "PPrf_MAIN".ON_WORK.A0301_A0302.Bordatrice.VelOvr_PLen_UpTo_3500;
       #ValueVelOvr[7] := "PPrf_MAIN".ON_WORK.A0301_A0302.Bordatrice.VelOvr_PLen_UpTo_4000;
       #ValueVelOvr[8] := "PPrf_MAIN".ON_WORK.A0301_A0302.Bordatrice.VelOvr_PLen_UpTo_4500;
       #ValueVelOvr[9] := "PPrf_MAIN".ON_WORK.A0301_A0302.Bordatrice.VelOvr_PLen_UpTo_5000;
       #ValueVelOvr[10] := "PPrf_MAIN".ON_WORK.A0301_A0302.Bordatrice.VelOvr_PLen_UpTo_5500;

       // Ciclo per verificare la variabile maggiore per prenderla in lavoro
       FOR #i := 1 TO 10 DO
           IF #ValueVelOvr[#i] >= #VelOvr_Max THEN
               #VelOvr_Max := #ValueVelOvr[#i];
           END_IF;
       END_FOR;// 
   END_REGION ;

   IF #VelOvr_Max = 0.0 THEN
       #VelOvr_Max := 100.0;
   END_IF;

   // *****************************************************************************************
   REGION // CALCOLO DELLA VELOCITA' E TRASFERIMENTO IN BASE ALLO STATO IMPIANTO

       #Ax.CIn.VelocityOverride.Enable := TRUE;
       //
       IF #Ax.CIn.Manager.Control_ON THEN

           IF #Ax.CIn.Manager.Control_ON THEN
               // CALCOLO VELOCITA' IN BASE ALL'OVERIDE
               #Ax.CIn.VelocityOverride.Value := #VelOvr_Max;
           ELSE
               #Ax.CIn.VelocityOverride.Value := 100.0;
           END_IF;

       END_IF;
   END_REGION ;
END_REGION

REGION Network 24 (SCL): [Ax] - CIn Manger
   // TRASFERIMENTO CIn MANAGER ALLA MACCHINA
   #Ax.CIn.Manager := #CIn.Manager.Ax;

   IF NOT #Ctrl.PosTargetEnable THEN
       #Ax.CIn.Manager.Pos := #Ctrl.Value.Ax_TargetLongPos;
   ELSE
       #Ax.CIn.Manager.Pos := #Ctrl.Value.PosTarget;
   END_IF;
END_REGION

REGION Network 25: [Ax] - Cin External alarm
   RUNG wire#powerrail
      Contact( FALSE )
      Coil( #Ax.CIn.ExternalAlarms )
   END_RUNG
   // the same network as SCL:
   #Ax.CIn.ExternalAlarms := FALSE;
END_REGION

REGION Network 26: [Ax] - Cin Ext Enable
   RUNG wire#powerrail
      Contact( TRUE )
      Coil( #Ax.CIn.Minus_ExtEnable )
   END_RUNG
   RUNG wire#powerrail
      "M_CmpGT"(Xa := #Ax.COut.ActualPosition, Xb := #Ax.CIn.Manager.Pos, MODULE := #Module, Ret_Val => #PositioningStop)
   END_RUNG
   RUNG wire#powerrail
      Contact( #CIn.CarroPareggCoda.BattutaVerticale.Rest )
      wire#w1
      Coil( #Ax.CIn.Plus_ExtEnable )
   END_RUNG
   RUNG wire#powerrail
      Contact( #CIn.CarroPareggCoda.BattutaVerticale.Work )
      I_Contact( #PositioningStop )
      Contact( #Ctrl.PosTargetEnable )
   END_RUNG wire#w1
   RUNG wire#powerrail
      Contact( #CIn.CarroPareggCoda.BattutaVerticale.Work )
      I_Contact( #CIn.CarroPareggCoda.Sens.FTC_Ingombro_In )
   END_RUNG wire#w1
   RUNG wire#powerrail
      Contact( #AreaInterface.Man )
      I_Contact( #CIn.Manager.Ax.Control_ON )
      Contact( #Sts.OP_CanMoveFreely )
   END_RUNG wire#w1
   // the same network as SCL:
   #Ax.CIn.Minus_ExtEnable := TRUE;
   #PositioningStop := "M_CmpGT"(Xa := #Ax.COut.ActualPosition, Xb := #Ax.CIn.Manager.Pos, MODULE := #Module);
   #Ax.CIn.Plus_ExtEnable := #CIn.CarroPareggCoda.BattutaVerticale.Rest OR (#CIn.CarroPareggCoda.BattutaVerticale.Work AND NOT #PositioningStop AND #Ctrl.PosTargetEnable) OR (#CIn.CarroPareggCoda.BattutaVerticale.Work AND NOT #CIn.CarroPareggCoda.Sens.FTC_Ingombro_In) OR (#AreaInterface.Man AND NOT #CIn.Manager.Ax.Control_ON AND #Sts.OP_CanMoveFreely);
END_REGION

REGION Network 27: [Ax] - Positioning Manager
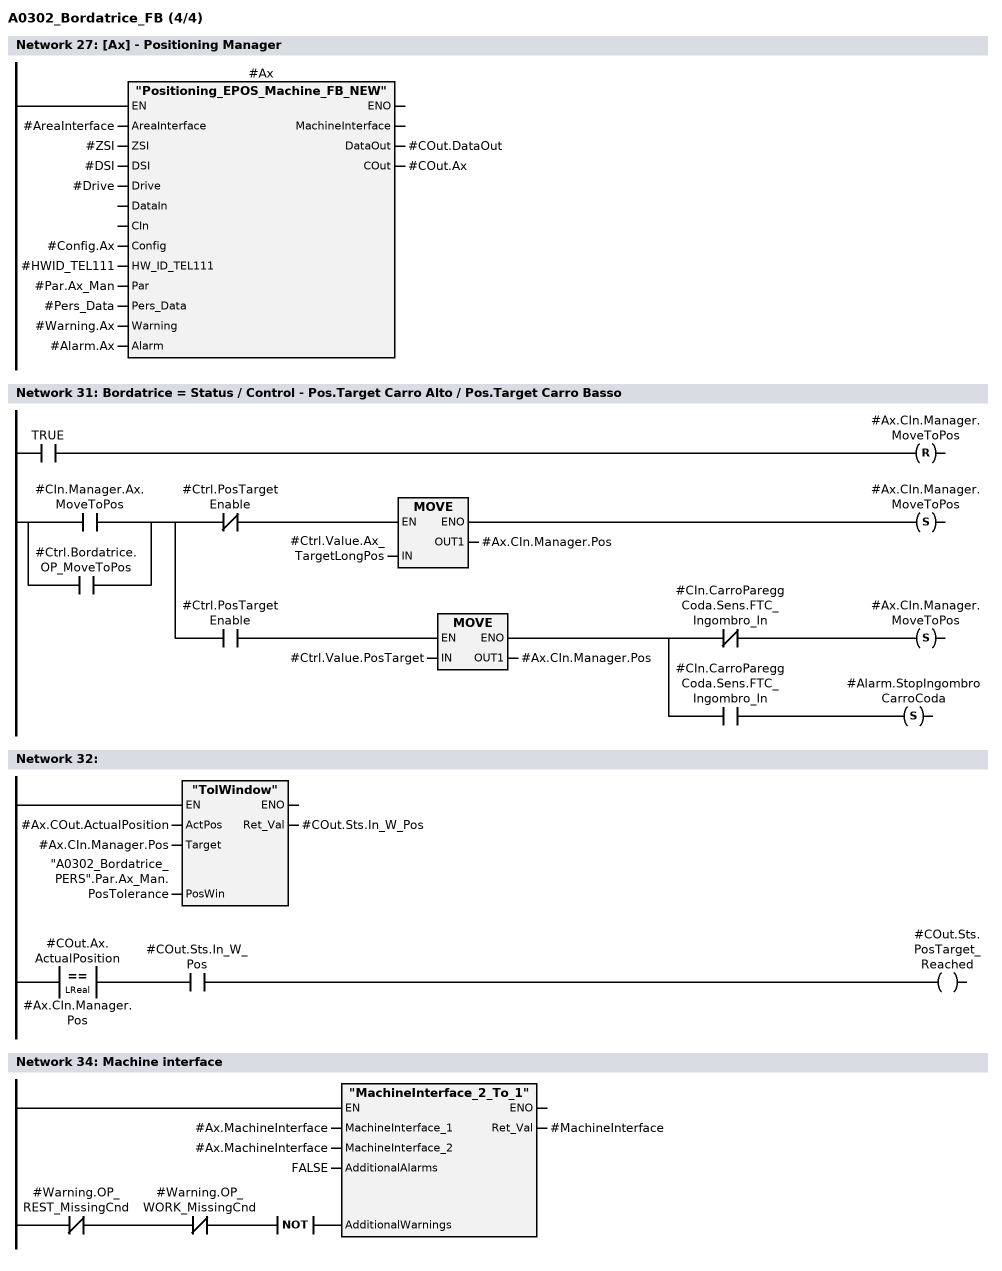
   RUNG wire#powerrail
      #Ax(AreaInterface := #AreaInterface, ZSI := #ZSI, DSI := #DSI, Drive := #Drive, DataIn :=, CIn :=, Config := #Config.Ax, HW_ID_TEL111 := #HWID_TEL111, Par := #Par.Ax_Man, Pers_Data := #Pers_Data, Warning := #Warning.Ax, Alarm := #Alarm.Ax, MachineInterface =>, DataOut => #COut.DataOut, COut => #COut.Ax)
   END_RUNG
   // the same network as SCL:
   #Ax(AreaInterface := #AreaInterface,   // "Positioning_EPOS_Machine_FB_NEW"
       ZSI := #ZSI,
       DSI := #DSI,
       Drive := #Drive,
       Config := #Config.Ax,
       HW_ID_TEL111 := #HWID_TEL111,
       Par := #Par.Ax_Man,
       Pers_Data := #Pers_Data,
       Warning := #Warning.Ax,
       Alarm := #Alarm.Ax,
       DataOut => #COut.DataOut,
       COut => #COut.Ax);
END_REGION

REGION Network 28: <+>
END_REGION

REGION Network 30: <<< CONTROLLO REQ da TRAKING E CAMBIO POS. >>>
END_REGION

REGION Network 31: Bordatrice = Status / Control - Pos.Target Carro Alto / Pos.Target Carro Basso
   RUNG wire#powerrail
      Contact( TRUE )
      R_Coil( #Ax.CIn.Manager.MoveToPos )
   END_RUNG
   RUNG wire#powerrail
      Contact( #CIn.Manager.Ax.MoveToPos )
      wire#w1
      I_Contact( #Ctrl.PosTargetEnable )
      Move(in := #Ctrl.Value.Ax_TargetLongPos, out1 => #Ax.CIn.Manager.Pos)
      S_Coil( #Ax.CIn.Manager.MoveToPos )
   END_RUNG
   RUNG wire#powerrail
      Contact( #Ctrl.Bordatrice.OP_MoveToPos )
   END_RUNG wire#w1
   RUNG wire#w1
      Contact( #Ctrl.PosTargetEnable )
      Move(in := #Ctrl.Value.PosTarget, out1 => #Ax.CIn.Manager.Pos)
      wire#w2
      I_Contact( #CIn.CarroPareggCoda.Sens.FTC_Ingombro_In )
      S_Coil( #Ax.CIn.Manager.MoveToPos )
   END_RUNG
   RUNG wire#w2
      Contact( #CIn.CarroPareggCoda.Sens.FTC_Ingombro_In )
      S_Coil( #Alarm.StopIngombroCarroCoda )
   END_RUNG
   // the same network as SCL:
   IF TRUE THEN #Ax.CIn.Manager.MoveToPos := FALSE; END_IF;
   #_w1 := #CIn.Manager.Ax.MoveToPos OR #Ctrl.Bordatrice.OP_MoveToPos;
   IF #_w1 AND NOT #Ctrl.PosTargetEnable THEN
       #Ax.CIn.Manager.Pos := #Ctrl.Value.Ax_TargetLongPos;
       #Ax.CIn.Manager.MoveToPos := TRUE;
   END_IF;
   #_w2 := #_w1 AND #Ctrl.PosTargetEnable;
   IF #_w2 THEN #Ax.CIn.Manager.Pos := #Ctrl.Value.PosTarget; END_IF;
   IF #_w2 AND NOT #CIn.CarroPareggCoda.Sens.FTC_Ingombro_In THEN #Ax.CIn.Manager.MoveToPos := TRUE; END_IF;
   IF #_w2 AND #CIn.CarroPareggCoda.Sens.FTC_Ingombro_In THEN #Alarm.StopIngombroCarroCoda := TRUE; END_IF;
END_REGION

REGION Network 32
   RUNG wire#powerrail
      "TolWindow"(ActPos := #Ax.COut.ActualPosition, Target := #Ax.CIn.Manager.Pos, PosWin := "A0302_Bordatrice_PERS".Par.Ax_Man.PosTolerance, Ret_Val => #COut.Sts.In_W_Pos)
   END_RUNG
   RUNG wire#powerrail
      { S7_Templates := "SrcType := LReal" } EQ_Contact(in1 := #COut.Ax.ActualPosition, in2 := #Ax.CIn.Manager.Pos)
      Contact( #COut.Sts.In_W_Pos )
      Coil( #COut.Sts.PosTarget_Reached )
   END_RUNG
   // the same network as SCL:
   #COut.Sts.In_W_Pos := "TolWindow"(ActPos := #Ax.COut.ActualPosition,
                           Target := #Ax.CIn.Manager.Pos,
                           PosWin := "A0302_Bordatrice_PERS".Par.Ax_Man.PosTolerance);
   #COut.Sts.PosTarget_Reached := (#COut.Ax.ActualPosition = #Ax.CIn.Manager.Pos) AND #COut.Sts.In_W_Pos;
END_REGION

REGION Network 33: << MAIN MACHINE STATUS >>
END_REGION

REGION Network 34: Machine interface
   RUNG wire#powerrail
      "MachineInterface_2_To_1"(AdditionalWarnings := wire#w1, MachineInterface_1 := #Ax.MachineInterface, MachineInterface_2 := #Ax.MachineInterface, AdditionalAlarms := FALSE, Ret_Val => #MachineInterface)
   END_RUNG
   RUNG wire#powerrail
      I_Contact( #Warning.OP_REST_MissingCnd )
      I_Contact( #Warning.OP_WORK_MissingCnd )
      Not()
   END_RUNG wire#w1
   // the same network as SCL:
   #MachineInterface := "MachineInterface_2_To_1"(MachineInterface_1 := #Ax.MachineInterface,
                           MachineInterface_2 := #Ax.MachineInterface,
                           AdditionalAlarms := FALSE,
                           AdditionalWarnings := NOT (NOT #Warning.OP_REST_MissingCnd AND NOT #Warning.OP_WORK_MissingCnd));
END_REGION
END_FUNCTION_BLOCK

FUNCTION_BLOCK "Lubr_Bordat"   // FB121, LAD
// stored: MemoryReserve 100, SetENOAutomatically false
   VAR
      Ton_Stop : TON_TIME;
      Ton_Start : TON_TIME;
      Ctrl { S7_SetPoint := 'True'} : Bool;
      Abilita : Bool;
   END_VAR
BEGIN

REGION Network 1
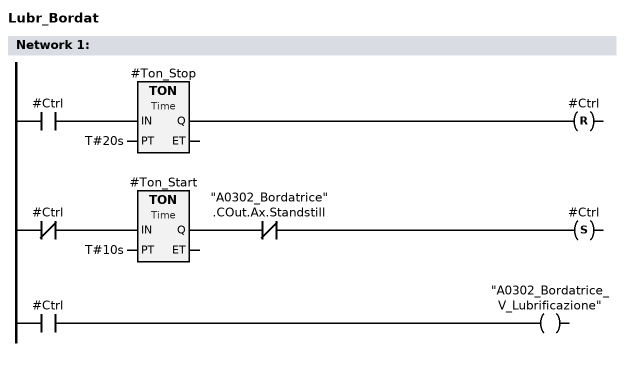
   RUNG wire#powerrail
      Contact( #Ctrl )
      { S7_Templates := "time_type := Time" } #Ton_Stop.TON(pt := T#20s, et =>)
      R_Coil( #Ctrl )
   END_RUNG
   RUNG wire#powerrail
      I_Contact( #Ctrl )
      { S7_Templates := "time_type := Time" } #Ton_Start.TON(pt := T#10s, et =>)
      I_Contact( "A0302_Bordatrice".COut.Ax.Standstill )
      S_Coil( #Ctrl )
   END_RUNG
   RUNG wire#powerrail
      Contact( #Ctrl )
      Coil( "A0302_Bordatrice_V_Lubrificazione" )
   END_RUNG
   // the same network as SCL:
   #Ton_Stop(IN := #Ctrl, PT := T#20s);   // TON
   IF #Ton_Stop.Q THEN #Ctrl := FALSE; END_IF;
   #Ton_Start(IN := NOT #Ctrl, PT := T#10s);   // TON
   IF #Ton_Start.Q AND NOT "A0302_Bordatrice".COut.Ax.Standstill THEN #Ctrl := TRUE; END_IF;
   "A0302_Bordatrice_V_Lubrificazione" := #Ctrl;
END_REGION
END_FUNCTION_BLOCK

FUNCTION "A0302_Rulliera_CALL" : Void   // FC136, LAD
// stored: SetENOAutomatically false
   VAR_TEMP
      Missing_Input : Bool;
      Missing_Output : Bool;
   END_VAR
   VAR CONSTANT
      MISSING : Int;
   END_VAR
BEGIN

REGION Network 1 (SCL): << TRASFERIMENTO stati CIn del blocco >>
   // SOSTITUIRE SYS BYPASS CON INGRESSI DIGITALI
   // TRASFERIMENTO COMANDI CIn MANAGER
   "A0302_Rulliera".CIn.Manager.Ax_1 := "A0302_Manager".COut.Rulliera.Ax_1;
   "A0302_Rulliera".CIn.Manager.Ax_2 := "A0302_Manager".COut.Rulliera.Ax_2;
   //
   "A0302_Rulliera".CIn.SemiAut_Pb := "A0302_Manager".DataIn.SemiAut_Pb;


   REGION TRASFERIMENTO STATI STAZIONE P5

       "A0302_Rulliera".CIn.Rulliera.Sollevamento := "A0301_Spintore_Lat".COut.Sollevatori;
       "A0302_Rulliera".CIn.P5.SpintoreLong := "A0302_Spintore".COut.Spintore;
       "A0302_Rulliera".CIn.P5.Sens := "A0302_Manager".CIn.P5.SpintoreLong.Sens;

   END_REGION ;

   REGION TRASFERIMENTO STATI RULLIERA dopo BORDATRICE

       "A0302_Rulliera".CIn.Rulliera.Centratori := "A0302_Centratori".COut.Centraggio;
       "A0302_Rulliera".CIn.Rulliera.Sollevamento := "A0302_Centratori".COut.Sollevamento;
       "A0302_Rulliera".CIn.Rulliera.Coda.Sens := "A0302_Manager".CIn.Rulliera.Coda.Sens;

       "A0302_Rulliera".CIn.CarroPareggCoda.Sens.FTC_Ingombro_In := "A0302_PareggiatoreCoda".IEC_FTC_Input.FTC_On;
       "A0302_Rulliera".CIn.CarroPareggCoda.Sens.FTC_Ingombro_Out := "A0302_PareggiatoreCoda".IEC_FTC_Output.FTC_On;
       "A0302_Rulliera".CIn.CarroPareggCoda.Sens.PresenzaMat := "A0302_PareggiatoreCoda".IEC_FTC_PresentMat.FTC_On;

   END_REGION ;

   REGION TRASFERIMENTO STATI CARRO PAREGGIATORE DI CODA

       "A0302_Rulliera".CIn.CarroPareggCoda.Ax := "A0302_PareggiatoreCoda".COut.Ax;
       "A0302_Rulliera".CIn.CarroPareggCoda.Bloccaggio := "A0302_PareggiatoreCoda".COut.Bloccaggio;
       "A0302_Rulliera".CIn.CarroPareggCoda.BattutaVerticale := "A0302_PareggiatoreCoda".COut.BattutaVerticale;
       "A0302_Rulliera".CIn.CarroPareggCoda.PareggiatoreLong := "A0302_PareggiatoreCoda".COut.PareggiatoreLong;
       "A0302_Rulliera".CIn.CarroPareggCoda.Sens:= "A0302_Manager".CIn.CarroPareggCoda.Sens;

   END_REGION ;

   REGION TRASFERIMENTO STATI CARRO PAREGGIATORE DI TESTA

       "A0302_Rulliera".CIn.CarroPareggTesta.Ax := "A0302_PareggiatoreTesta".COut.Ax;
       "A0302_Rulliera".CIn.CarroPareggTesta.Bloccaggio := "A0302_PareggiatoreTesta".COut.Bloccaggio;
       "A0302_Rulliera".CIn.CarroPareggTesta.Centraggio := "A0302_PareggiatoreTesta".COut.Centraggio;
       "A0302_Rulliera".CIn.CarroPareggTesta.Sollevatore := "A0302_PareggiatoreTesta".COut.Sollevatore;
       "A0302_Rulliera".CIn.CarroPareggTesta.Sens := "A0302_Manager".CIn.CarroPareggTesta.Sens;

   END_REGION ;

   // TRASFERIMENTO STATO DELLE ZONE INGRESSO E USCITA DELLA STAZIONE
   "A0302_Rulliera".CIn.BTrk.ZoneA0302Entry_Empty := "A0302_Manager".Sts.BTrk.ZoneA0302Entry_Empty;
   "A0302_Rulliera".CIn.BTrk.ZoneA0302Exit_Empty := "A0302_Manager".Sts.BTrk.ZoneA0302Exit_Empty;
END_REGION

REGION Network 2 (SCL): <<< Data In >>>
END_REGION

REGION Network 3 (SCL): Data In- SENSORI
   // INGRESSI SENSORI RULLIERA
   //
   "A0302_Rulliera".DataIn.Sens.Coda.FTC_Rall := "A0302_Rulliera_Lato_2_Coda_Phc_1_ControlloNuovoPezzo";
   "A0302_Rulliera".DataIn.Sens.Coda.FTC_Prox_Ing := "A0302_Rulliera_Lato_2_Coda_Phc_2_ControlloNuovoPezzo";
   // [%I351.7] "A0302_Rulliera_Lato_1_Testa_Phc_PezzoCentraturaCentrale";
   // [%I303.0] "A0302_Rulliera_Lato_2_Coda_Phc_2_ControlloNuovoPezzo"
   "A0302_Rulliera".DataIn.Sens.Centro.FTC_Centrale := "A0302_Rulliera_Lato_1_Testa_Phc_PezzoCentraturaCentrale";
   //
END_REGION

REGION Network 4: DataIn
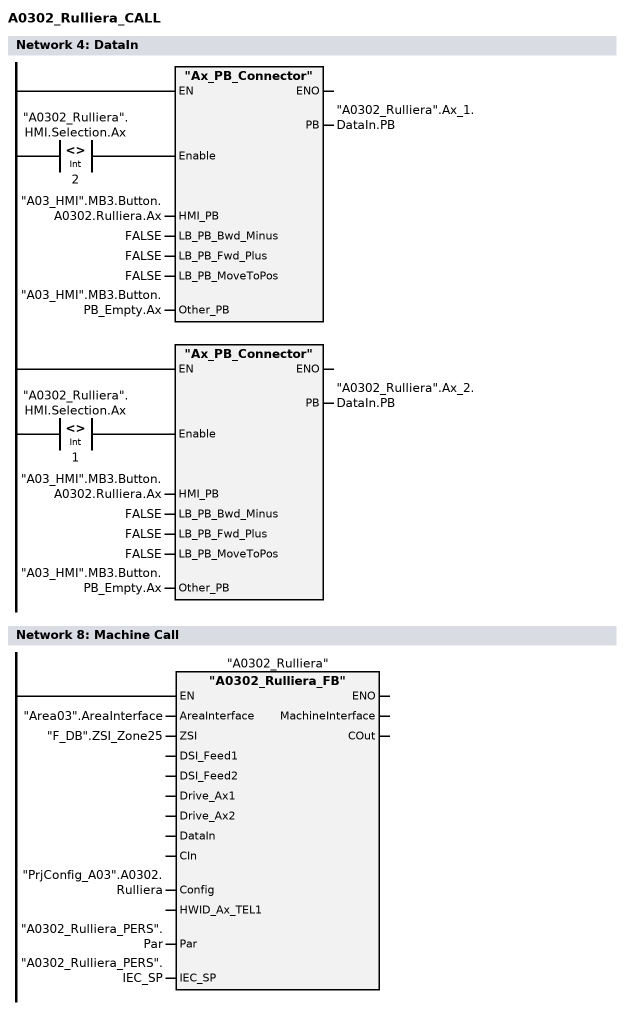
   RUNG wire#powerrail
      "Ax_PB_Connector"(Enable := wire#w1, HMI_PB := "A03_HMI".MB3.Button.A0302.Rulliera.Ax, LB_PB_Bwd_Minus := FALSE, LB_PB_Fwd_Plus := FALSE, LB_PB_MoveToPos := FALSE, Other_PB := "A03_HMI".MB3.Button.PB_Empty.Ax, PB => "A0302_Rulliera".Ax_1.DataIn.PB)
   END_RUNG
   RUNG wire#powerrail
      { S7_Templates := "SrcType := Int" } NE_Contact(in1 := "A0302_Rulliera".HMI.Selection.Ax, in2 := 2)
   END_RUNG wire#w1
   RUNG wire#powerrail
      "Ax_PB_Connector"(Enable := wire#w2, HMI_PB := "A03_HMI".MB3.Button.A0302.Rulliera.Ax, LB_PB_Bwd_Minus := FALSE, LB_PB_Fwd_Plus := FALSE, LB_PB_MoveToPos := FALSE, Other_PB := "A03_HMI".MB3.Button.PB_Empty.Ax, PB => "A0302_Rulliera".Ax_2.DataIn.PB)
   END_RUNG
   RUNG wire#powerrail
      { S7_Templates := "SrcType := Int" } NE_Contact(in1 := "A0302_Rulliera".HMI.Selection.Ax, in2 := 1)
   END_RUNG wire#w2
   // the same network as SCL:
   "Ax_PB_Connector"(Enable := "A0302_Rulliera".HMI.Selection.Ax <> 2,
                     HMI_PB := "A03_HMI".MB3.Button.A0302.Rulliera.Ax,
                     LB_PB_Bwd_Minus := FALSE,
                     LB_PB_Fwd_Plus := FALSE,
                     LB_PB_MoveToPos := FALSE,
                     Other_PB := "A03_HMI".MB3.Button.PB_Empty.Ax,
                     PB => "A0302_Rulliera".Ax_1.DataIn.PB);
   "Ax_PB_Connector"(Enable := "A0302_Rulliera".HMI.Selection.Ax <> 1,
                     HMI_PB := "A03_HMI".MB3.Button.A0302.Rulliera.Ax,
                     LB_PB_Bwd_Minus := FALSE,
                     LB_PB_Fwd_Plus := FALSE,
                     LB_PB_MoveToPos := FALSE,
                     Other_PB := "A03_HMI".MB3.Button.PB_Empty.Ax,
                     PB => "A0302_Rulliera".Ax_2.DataIn.PB);
END_REGION

REGION Network 5 (SCL): DSI
   // Di solito facciamo struct DSI con dentro Rulliera 1 / Rulliera 2

   "A0302_Rulliera".DSI_Feed1 := "F_DB".DSI_Rulliera1;
   "A0302_Rulliera".DSI_Feed2 := "F_DB".DSI_Rulliera2;
END_REGION

REGION Network 6 (SCL): Drive
   // Anche qui di solito c'è una struttura Drive con dentro 2 membri
   // 

   "A0302_Rulliera".Drive_Ax1.Infeed_ON := "Areas_ITF".AG.Infeed_Running;;
   "A0302_Rulliera".Drive_Ax1.AccessPoint := "HW_Const_Values".CU6_PN_605A1_ModuleAccessPoint;
   "A0302_Rulliera".Drive_Ax1.AxisID := "CU6_ID_2_1990A1_1_1990M1";
   "A0302_Rulliera".Drive_Ax1.TokenChain := "TOKENCHAIN_CU6";

   "A0302_Rulliera".Drive_Ax2.Infeed_ON := "Areas_ITF".AG.Infeed_Running;
   "A0302_Rulliera".Drive_Ax2.AccessPoint := "HW_Const_Values".CU6_PN_605A1_ModuleAccessPoint;
   "A0302_Rulliera".Drive_Ax2.AxisID := "CU6_ID_3_1990A1_2_2000M1";
   "A0302_Rulliera".Drive_Ax2.TokenChain := "TOKENCHAIN_CU6";
END_REGION

REGION Network 7 (SCL): HW
   "A0302_Rulliera".HWID_Ax_TEL1[1] := "HW_Const_Values".CU6_PN_1990A1_1_Standard_telegram_1;

   "A0302_Rulliera".HWID_Ax_TEL1[2] := "HW_Const_Values".CU6_PN_1990A1_2_Standard_telegram_1;
END_REGION

REGION Network 8: Machine Call
   RUNG wire#powerrail
      "A0302_Rulliera"(AreaInterface := "Area03".AreaInterface, ZSI := "F_DB".ZSI_Zone25, DSI_Feed1 :=, DSI_Feed2 :=, Drive_Ax1 :=, Drive_Ax2 :=, DataIn :=, CIn :=, Config := "PrjConfig_A03".A0302.Rulliera, HWID_Ax_TEL1 :=, Par := "A0302_Rulliera_PERS".Par, IEC_SP := "A0302_Rulliera_PERS".IEC_SP, MachineInterface =>, COut =>)
   END_RUNG
   // the same network as SCL:
   "A0302_Rulliera"(AreaInterface := "Area03".AreaInterface,   // "A0302_Rulliera_FB"
                    ZSI := "F_DB".ZSI_Zone25,
                    Config := "PrjConfig_A03".A0302.Rulliera,
                    Par := "A0302_Rulliera_PERS".Par,
                    IEC_SP := "A0302_Rulliera_PERS".IEC_SP);
END_REGION
END_FUNCTION

FUNCTION_BLOCK "A0302_Rulliera_FB"   // FB64, LAD
// stored: MemoryReserve 100, SetENOAutomatically false
   VAR_INPUT
      AreaInterface : "AreaInterface";
      ZSI : "udt_ZoneSafetyInterface";
      DSI_Feed1 : "udt_DeviceSafetyInterface";
      DSI_Feed2 : "udt_DeviceSafetyInterface";
      Drive_Ax1 : "TAx_DriveInterface";
      Drive_Ax2 : "TAx_DriveInterface";
      DataIn : Struct
         Ax : "SpeedMachine_DataIn";
         Sens : Struct
            Coda { ExternalAccessible := 'False'; ExternalVisible := 'False'; ExternalWritable := 'False'} : Struct
               FTC_Rall : Bool;   // Sensori presenza materiale banco rallentamento ingresso
               FTC_Prox_Ing : Bool;   // Sensori presenza materiale banco limite ingresso
            END_STRUCT;
            Centro { ExternalAccessible := 'False'; ExternalVisible := 'False'; ExternalWritable := 'False'} : Struct
               FTC_Centrale : Bool;
            END_STRUCT;
         END_STRUCT;
      END_STRUCT;
      CIn { ExternalAccessible := 'False'; ExternalVisible := 'False'; ExternalWritable := 'False'} : Struct
         Manager : Struct
            Ax_1 : "SpeedMachine_CIn_Manager";
            Ax_2 : "SpeedMachine_CIn_Manager";
         END_STRUCT;
         SemiAut_Pb : Bool;
         P5 : Struct
            Sollevatori : "ValveMachine_COut";
            SpintoreLong : "ValveMachine_COut";
            Sens : Struct
               FTC_Ingombro_A0301 : Bool;   // 1614BF1 - I50.7
            END_STRUCT;
         END_STRUCT;
         Bordatrice : Struct
            StopBordatrice : Bool;   // Stop Bordatrice da controllo quota spazio rimanente su rulliera di coda
            ReadyForMove : Bool;   // Pronto al movimento
            StandbyBordatrice : Bool;
         END_STRUCT;
         Rulliera : Struct
            Centratori : "ValveMachine_COut";   // Chiusura Centratori
            Sollevamento : "ValveMachine_COut";   // Solleva centratori
            Coda : Struct
               Sens : Struct
                  FTC_Rall : Bool;   // Sensori presenza materiale banco rallentamento ingresso
                  FTC_Prox_Ing : Bool;   // Sensori presenza materiale banco limite ingresso
               END_STRUCT;
            END_STRUCT;
            Centro : Struct
               Sens : Struct
                  FTC_Centrale : Bool;   // 2010BF1 - I50.2
               END_STRUCT;
            END_STRUCT;
         END_STRUCT;
         CarroPareggCoda : Struct
            Ax : "Positioning_DOL_Machine_COut";
            Bloccaggio : "ValveMachine_COut";
            BattutaVerticale : "ValveMachine_COut";
            PareggiatoreLong : "ValveMachine_COut";
            Sens : Struct
               FTC_Ingombro_In : Bool;   // 2012BF1 - I50.0
               FTC_Ingombro_Out : Bool;   // 2012BF2 - I50.1
               PresenzaMat : Bool;   // FC presenza materiale agganciato lato paregg coda
               PosPareggLong : Struct
                  Value : LReal;
                  CheckMeasure : Bool;
                  Standstill : Bool;
               END_STRUCT;
            END_STRUCT;
         END_STRUCT;
         CarroPareggTesta : Struct
            Ax : "Positioning_DOL_Machine_COut";
            Bloccaggio : "ValveMachine_COut";
            Centraggio : "ValveMachine_COut";
            Sollevatore : "ValveMachine_COut";
            Sens : Struct
               FTC1_Rall : Bool;   // 2010BF2 - I50.3
               FTC2_Prox_Ls : Bool;   // 2010BF3 - I50.4
               PresenzaMat : Bool;   // FC presenza materiale agganciato lato paregg testa
            END_STRUCT;
         END_STRUCT;
         BTrk : Struct
            ZoneA0302Entry_Empty : Bool;
            ZoneA0302Exit_Empty : Bool;
         END_STRUCT;
      END_STRUCT;
      Config : Struct
         Ax : "SpeedMachine_Config";
      END_STRUCT;
      HWID_Ax_TEL1 : Array[1..2] of HW_SUBMODULE;
   END_VAR
   VAR_OUTPUT
      MachineInterface : "MachineInterface";
      COut : Struct
         Ax_1 : "SpeedMachine_COut";
         Ax_2 : "SpeedMachine_COut";
         Ax_VelOveride : Struct
            Enable : Bool;
            Value : Real;
         END_STRUCT;
      END_STRUCT;
   END_VAR
   VAR_IN_OUT
      Par : Struct
         Ax : "SpeedMachine_Par";
         Ax_Aut : "A0301_Mach_Speed_Par";
      END_STRUCT;
      IEC_SP : Struct
         FTC_CodaRall : Struct
            TON_PT : Time;
            TOF_PT : Time;
         END_STRUCT;
         FTC_CodaProx_Ing : Struct
            TON_PT : Time;
            TOF_PT : Time;
         END_STRUCT;
         FTC_Centro : Struct
            TON_PT : Time;
            TOF_PT : Time;
         END_STRUCT;
      END_STRUCT;
   END_VAR
   VAR
      Alarm : Struct
         Rulliera : Array[1..2] of "SpeedMachine_Alr";
      END_STRUCT;
      Warning : Struct
         Rulliera : Array[1..2] of "SpeedMachine_Wng";
         OP_REST_MissingCnd : Bool;   // Mancanza comando arresto
         OP_WORK_MissingCnd : Bool;   // Mancanza consenso lavoro
      END_STRUCT;
      HMI : Struct
         Selection : Struct   // 0=Disable / 1=Enable Pin
            Ax : Int;   // 0:Entrambe / 1:Rulliera Ax1 / 2:Rulliera Ax2
         END_STRUCT;
      END_STRUCT;
      Ax_1 : "SpeedMachine_FB";
      Ax_2 : "SpeedMachine_FB";
      ValueVelOvr { ExternalAccessible := 'False'; ExternalVisible := 'False'; ExternalWritable := 'False'} : Array[1..10] of Real;
      Sts : Struct
         OP_CanMoveFreely : Bool;
         OP_Bwd_Cnd : Bool;
         OP_Fwd_Cnd : Bool;
      END_STRUCT;
      Ctrl : Struct
         OP_Bwd_Man : Bool;
         OP_Fwd_Man : Bool;
         OP_Bwd_Aut : Bool;
         OP_Fwd_Aut : Bool;
         OP_Bwd_Run : Bool;
         OP_Fwd_Run : Bool;
      END_STRUCT;
      AUX : Struct
         OP_Bwd_PB : Bool;
         OP_Fwd_PB : Bool;
      END_STRUCT;
      TON_OP_REST_MissingCnd { S7_SetPoint := 'True'} : TON_TIME;
      TON_OP_WORK_MissingCnd { S7_SetPoint := 'True'} : TON_TIME;
      IEC_FTC_CodaRall : Struct
         TON_Delay : IEC_TIMER;
         TOF_Delay { S7_SetPoint := 'True'} : IEC_TIMER;
         FTC_On { S7_SetPoint := 'True'} : Bool;
      END_STRUCT;
      IEC_FTC_CodaProxIng : Struct
         TON_Delay : IEC_TIMER;
         TOF_Delay { S7_SetPoint := 'True'} : IEC_TIMER;
         FTC_On { S7_SetPoint := 'True'} : Bool;
      END_STRUCT;
      IEC_FTC_Centro : Struct
         TON_Delay : IEC_TIMER;
         TOF_Delay { S7_SetPoint := 'True'} : IEC_TIMER;
         FTC_On { S7_SetPoint := 'True'} : Bool;
      END_STRUCT;
   END_VAR
   VAR_TEMP
      PE : Struct
         OP_Bwd_PB : Bool;
         OP_Fwd_PB : Bool;
      END_STRUCT;
      VelOvr_Max : Real;   // Velocità max trovata
      i : Int;
      Check : Struct
         Cndz1_StartFwd : Bool;   // Check conditions to P4
         Cndz2_StartFwd : Bool;   // Check conditions to Allineatore laterale
      END_STRUCT;
   END_VAR
   VAR_TEMP   // added for the SCL form of the ladder/FBD networks
      _w1 : Bool;
      _w2 : Bool;
      _w3 : Bool;
   END_VAR
BEGIN

REGION Network 1 (SCL): == Riferimenti [Ax] - Speed Machine ==
   // ******************************************************************************************
   REGION // TRASFERIMENTO DELLE RAMPE

       // Rampe in Manuale
       IF #AreaInterface.Man AND NOT #CIn.SemiAut_Pb THEN
           #Ax_1.CIn.Manager.Vel := #Ax_2.CIn.Manager.Vel := #Par.Ax.Man.VelFwdHigh;
           #Ax_1.CIn.Manager.Acc :=  #Ax_2.CIn.Manager.Acc := #Par.Ax.Man.Acc;
           #Ax_1.CIn.Manager.Dec := #Ax_2.CIn.Manager.Dec := #Par.Ax.Man.Dec;
       END_IF;
   END_REGION

   // ******************************************************************************************
   REGION // CALCOLO DELLA VELOCITA' TRASFERITA DALL'IMPIANTO IN BASE ALLA LUNGHEZZA DEL PEZZO 

       // Inizializzo variabile di appoggio controllo overide massimo a un valore basso rispetto setpoint
       IF "Sys".AuxFirstPLCCycle THEN
           #VelOvr_Max := 100.0;
       END_IF;

       // Trasferisco le varibili su un array
       #ValueVelOvr[1] := "PPrf_MAIN".ON_WORK.A0301_A0302.Trasporto.VelOvr_PLen_UpTo_1000;
       #ValueVelOvr[2] := "PPrf_MAIN".ON_WORK.A0301_A0302.Trasporto.VelOvr_PLen_UpTo_1500;
       #ValueVelOvr[3] := "PPrf_MAIN".ON_WORK.A0301_A0302.Trasporto.VelOvr_PLen_UpTo_2000;
       #ValueVelOvr[4] := "PPrf_MAIN".ON_WORK.A0301_A0302.Trasporto.VelOvr_PLen_UpTo_2500;
       #ValueVelOvr[5] := "PPrf_MAIN".ON_WORK.A0301_A0302.Trasporto.VelOvr_PLen_UpTo_3000;
       #ValueVelOvr[6] := "PPrf_MAIN".ON_WORK.A0301_A0302.Trasporto.VelOvr_PLen_UpTo_3500;
       #ValueVelOvr[7] := "PPrf_MAIN".ON_WORK.A0301_A0302.Trasporto.VelOvr_PLen_UpTo_4000;
       #ValueVelOvr[8] := "PPrf_MAIN".ON_WORK.A0301_A0302.Trasporto.VelOvr_PLen_UpTo_4500;
       #ValueVelOvr[9] := "PPrf_MAIN".ON_WORK.A0301_A0302.Trasporto.VelOvr_PLen_UpTo_5000;
       #ValueVelOvr[10] := "PPrf_MAIN".ON_WORK.A0301_A0302.Trasporto.VelOvr_PLen_UpTo_5500;


       // Ciclo per verificare la variabile maggiore per prenderla in lavoro
       FOR #i := 1 TO 10 DO
           IF #ValueVelOvr[#i] >= #VelOvr_Max THEN
               #VelOvr_Max := #ValueVelOvr[#i];
           END_IF;
       END_FOR;
   END_REGION ;

   IF #VelOvr_Max = 0.0 THEN
       #VelOvr_Max := 100.0;
   END_IF;

   // ******************************************************************************************
   REGION // CALCOLO DELLA VELOCITA' E TRASFERIMENTO IN BASE ALLO STATO IMPIANTO

       #Ax_1.CIn.VelocityOverride.Enable := TRUE;
       #Ax_2.CIn.VelocityOverride.Enable := TRUE;

       IF #Ax_1.CIn.Manager.Control_ON THEN
           // CALCOLO VELOCITA' IN BASE ALL'OVERIDE
           #Ax_1.CIn.VelocityOverride.Value :=  #VelOvr_Max;
       ELSE
           #Ax_1.CIn.VelocityOverride.Value := 100.0;
           END_IF;

           IF #Ax_2.CIn.Manager.Control_ON THEN
               #Ax_2.CIn.VelocityOverride.Value := #VelOvr_Max;
           ELSE
               #Ax_2.CIn.VelocityOverride.Value := 100.0;
           END_IF;
       END_REGION ;
END_REGION

REGION Network 3: DataIn - FTC CodaRall
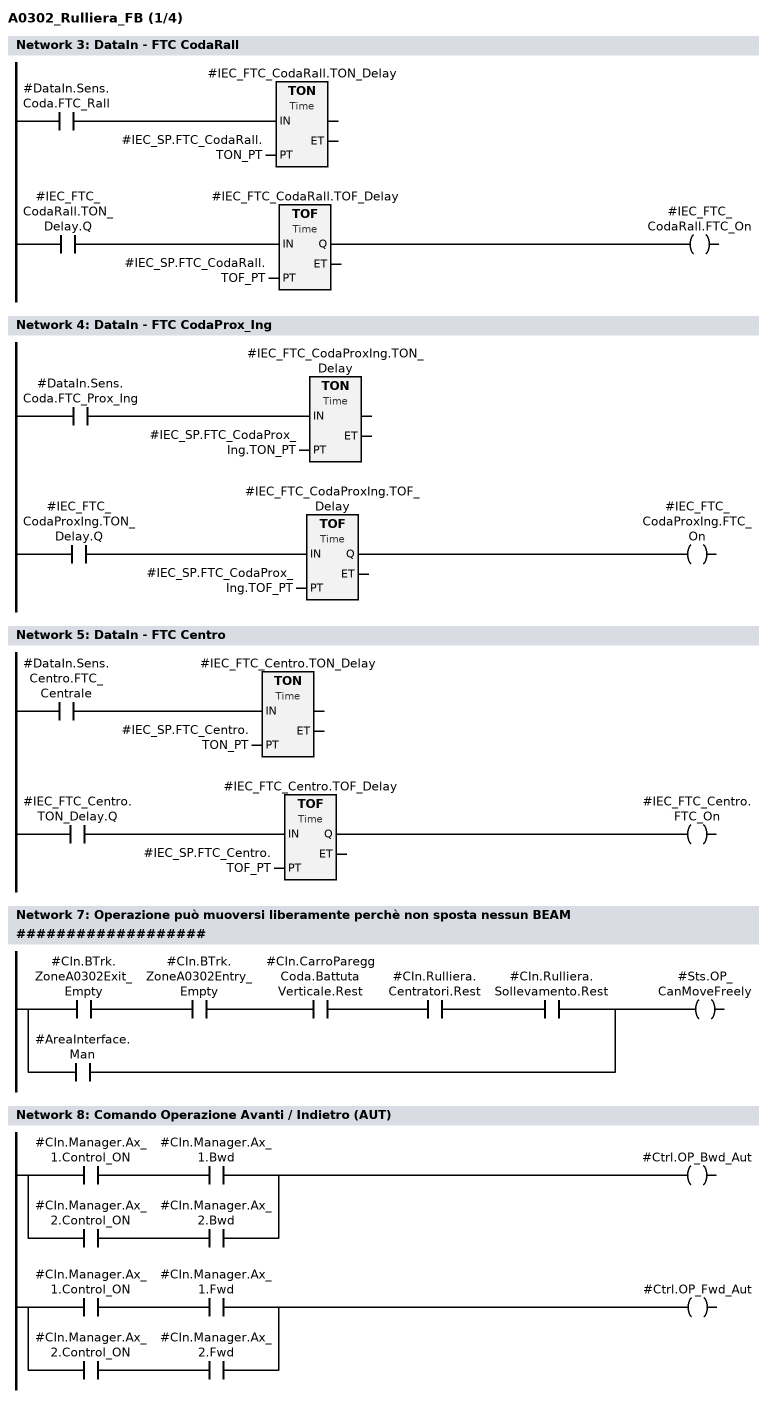
   RUNG wire#powerrail
      Contact( #DataIn.Sens.Coda.FTC_Rall )
      { S7_Templates := "time_type := Time" } #IEC_FTC_CodaRall.TON_Delay.TON(pt := #IEC_SP.FTC_CodaRall.TON_PT, et =>)
   END_RUNG
   RUNG wire#powerrail
      Contact( #IEC_FTC_CodaRall.TON_Delay.Q )
      { S7_Templates := "time_type := Time" } #IEC_FTC_CodaRall.TOF_Delay.TOF(pt := #IEC_SP.FTC_CodaRall.TOF_PT, et =>)
      Coil( #IEC_FTC_CodaRall.FTC_On )
   END_RUNG
   // the same network as SCL:
   #IEC_FTC_CodaRall.TON_Delay.TON(IN := #DataIn.Sens.Coda.FTC_Rall, PT := #IEC_SP.FTC_CodaRall.TON_PT);
   #IEC_FTC_CodaRall.TOF_Delay.TOF(IN := #IEC_FTC_CodaRall.TON_Delay.Q, PT := #IEC_SP.FTC_CodaRall.TOF_PT);
   #IEC_FTC_CodaRall.FTC_On := #IEC_FTC_CodaRall.TOF_Delay.Q;
END_REGION

REGION Network 4: DataIn - FTC CodaProx_Ing
   RUNG wire#powerrail
      Contact( #DataIn.Sens.Coda.FTC_Prox_Ing )
      { S7_Templates := "time_type := Time" } #IEC_FTC_CodaProxIng.TON_Delay.TON(pt := #IEC_SP.FTC_CodaProx_Ing.TON_PT, et =>)
   END_RUNG
   RUNG wire#powerrail
      Contact( #IEC_FTC_CodaProxIng.TON_Delay.Q )
      { S7_Templates := "time_type := Time" } #IEC_FTC_CodaProxIng.TOF_Delay.TOF(pt := #IEC_SP.FTC_CodaProx_Ing.TOF_PT, et =>)
      Coil( #IEC_FTC_CodaProxIng.FTC_On )
   END_RUNG
   // the same network as SCL:
   #IEC_FTC_CodaProxIng.TON_Delay.TON(IN := #DataIn.Sens.Coda.FTC_Prox_Ing,
                           PT := #IEC_SP.FTC_CodaProx_Ing.TON_PT);
   #IEC_FTC_CodaProxIng.TOF_Delay.TOF(IN := #IEC_FTC_CodaProxIng.TON_Delay.Q,
                           PT := #IEC_SP.FTC_CodaProx_Ing.TOF_PT);
   #IEC_FTC_CodaProxIng.FTC_On := #IEC_FTC_CodaProxIng.TOF_Delay.Q;
END_REGION

REGION Network 5: DataIn - FTC Centro
   RUNG wire#powerrail
      Contact( #DataIn.Sens.Centro.FTC_Centrale )
      { S7_Templates := "time_type := Time" } #IEC_FTC_Centro.TON_Delay.TON(pt := #IEC_SP.FTC_Centro.TON_PT, et =>)
   END_RUNG
   RUNG wire#powerrail
      Contact( #IEC_FTC_Centro.TON_Delay.Q )
      { S7_Templates := "time_type := Time" } #IEC_FTC_Centro.TOF_Delay.TOF(pt := #IEC_SP.FTC_Centro.TOF_PT, et =>)
      Coil( #IEC_FTC_Centro.FTC_On )
   END_RUNG
   // the same network as SCL:
   #IEC_FTC_Centro.TON_Delay.TON(IN := #DataIn.Sens.Centro.FTC_Centrale, PT := #IEC_SP.FTC_Centro.TON_PT);
   #IEC_FTC_Centro.TOF_Delay.TOF(IN := #IEC_FTC_Centro.TON_Delay.Q, PT := #IEC_SP.FTC_Centro.TOF_PT);
   #IEC_FTC_Centro.FTC_On := #IEC_FTC_Centro.TOF_Delay.Q;
END_REGION

REGION Network 7: Operazione può muoversi liberamente perchè non sposta nessun BEAM ###################
   RUNG wire#powerrail
      Contact( #CIn.BTrk.ZoneA0302Exit_Empty )
      Contact( #CIn.BTrk.ZoneA0302Entry_Empty )
      Contact( #CIn.CarroPareggCoda.BattutaVerticale.Rest )
      Contact( #CIn.Rulliera.Centratori.Rest )
      Contact( #CIn.Rulliera.Sollevamento.Rest )
      wire#w1
      Coil( #Sts.OP_CanMoveFreely )
   END_RUNG
   RUNG wire#powerrail
      Contact( #AreaInterface.Man )
   END_RUNG wire#w1
   // the same network as SCL:
   #Sts.OP_CanMoveFreely := (#CIn.BTrk.ZoneA0302Exit_Empty AND #CIn.BTrk.ZoneA0302Entry_Empty AND #CIn.CarroPareggCoda.BattutaVerticale.Rest AND #CIn.Rulliera.Centratori.Rest AND #CIn.Rulliera.Sollevamento.Rest) OR #AreaInterface.Man;
END_REGION

REGION Network 8: Comando Operazione Avanti / Indietro (AUT)
   RUNG wire#powerrail
      Contact( #CIn.Manager.Ax_1.Control_ON )
      Contact( #CIn.Manager.Ax_1.Bwd )
      wire#w1
      Coil( #Ctrl.OP_Bwd_Aut )
   END_RUNG
   RUNG wire#powerrail
      Contact( #CIn.Manager.Ax_2.Control_ON )
      Contact( #CIn.Manager.Ax_2.Bwd )
   END_RUNG wire#w1
   RUNG wire#powerrail
      Contact( #CIn.Manager.Ax_1.Control_ON )
      Contact( #CIn.Manager.Ax_1.Fwd )
      wire#w2
      Coil( #Ctrl.OP_Fwd_Aut )
   END_RUNG
   RUNG wire#powerrail
      Contact( #CIn.Manager.Ax_2.Control_ON )
      Contact( #CIn.Manager.Ax_2.Fwd )
   END_RUNG wire#w2
   // the same network as SCL:
   #Ctrl.OP_Bwd_Aut := (#CIn.Manager.Ax_1.Control_ON AND #CIn.Manager.Ax_1.Bwd) OR (#CIn.Manager.Ax_2.Control_ON AND #CIn.Manager.Ax_2.Bwd);
   #Ctrl.OP_Fwd_Aut := (#CIn.Manager.Ax_1.Control_ON AND #CIn.Manager.Ax_1.Fwd) OR (#CIn.Manager.Ax_2.Control_ON AND #CIn.Manager.Ax_2.Fwd);
END_REGION

REGION Network 9: Comando Operazione Lavoro / Riposo (MAN)
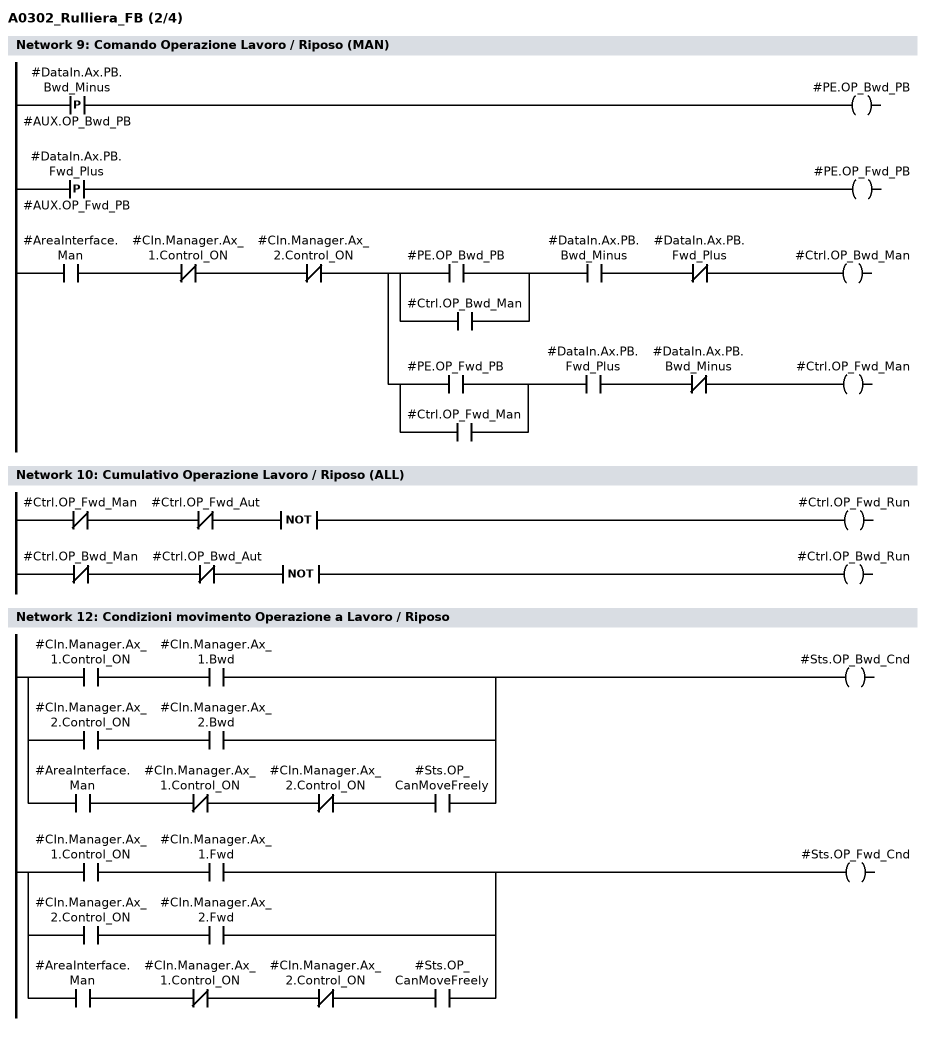
   RUNG wire#powerrail
      P_Contact(operand := #DataIn.Ax.PB.Bwd_Minus, bit := #AUX.OP_Bwd_PB)
      Coil( #PE.OP_Bwd_PB )
   END_RUNG
   RUNG wire#powerrail
      P_Contact(operand := #DataIn.Ax.PB.Fwd_Plus, bit := #AUX.OP_Fwd_PB)
      Coil( #PE.OP_Fwd_PB )
   END_RUNG
   RUNG wire#powerrail
      Contact( #AreaInterface.Man )
      I_Contact( #CIn.Manager.Ax_1.Control_ON )
      I_Contact( #CIn.Manager.Ax_2.Control_ON )
      wire#w1
      Contact( #PE.OP_Bwd_PB )
      wire#w2
      Contact( #DataIn.Ax.PB.Bwd_Minus )
      I_Contact( #DataIn.Ax.PB.Fwd_Plus )
      Coil( #Ctrl.OP_Bwd_Man )
   END_RUNG
   RUNG wire#w1
      Contact( #Ctrl.OP_Bwd_Man )
   END_RUNG wire#w2
   RUNG wire#w1
      Contact( #PE.OP_Fwd_PB )
      wire#w3
      Contact( #DataIn.Ax.PB.Fwd_Plus )
      I_Contact( #DataIn.Ax.PB.Bwd_Minus )
      Coil( #Ctrl.OP_Fwd_Man )
   END_RUNG
   RUNG wire#w1
      Contact( #Ctrl.OP_Fwd_Man )
   END_RUNG wire#w3
   // the same network as SCL:
   #_w1 := #DataIn.Ax.PB.Bwd_Minus AND NOT #AUX.OP_Bwd_PB;   // rising edge of #DataIn.Ax.PB.Bwd_Minus
   #AUX.OP_Bwd_PB := #DataIn.Ax.PB.Bwd_Minus;
   #PE.OP_Bwd_PB := #_w1;
   #_w2 := #DataIn.Ax.PB.Fwd_Plus AND NOT #AUX.OP_Fwd_PB;   // rising edge of #DataIn.Ax.PB.Fwd_Plus
   #AUX.OP_Fwd_PB := #DataIn.Ax.PB.Fwd_Plus;
   #PE.OP_Fwd_PB := #_w2;
   #_w3 := #AreaInterface.Man AND NOT #CIn.Manager.Ax_1.Control_ON AND NOT #CIn.Manager.Ax_2.Control_ON;
   #Ctrl.OP_Bwd_Man := #_w3 AND (#PE.OP_Bwd_PB OR #Ctrl.OP_Bwd_Man) AND #DataIn.Ax.PB.Bwd_Minus AND NOT #DataIn.Ax.PB.Fwd_Plus;
   #Ctrl.OP_Fwd_Man := #_w3 AND (#PE.OP_Fwd_PB OR #Ctrl.OP_Fwd_Man) AND #DataIn.Ax.PB.Fwd_Plus AND NOT #DataIn.Ax.PB.Bwd_Minus;
END_REGION

REGION Network 10: Cumulativo Operazione Lavoro / Riposo (ALL)
   RUNG wire#powerrail
      I_Contact( #Ctrl.OP_Fwd_Man )
      I_Contact( #Ctrl.OP_Fwd_Aut )
      Not()
      Coil( #Ctrl.OP_Fwd_Run )
   END_RUNG
   RUNG wire#powerrail
      I_Contact( #Ctrl.OP_Bwd_Man )
      I_Contact( #Ctrl.OP_Bwd_Aut )
      Not()
      Coil( #Ctrl.OP_Bwd_Run )
   END_RUNG
   // the same network as SCL:
   #Ctrl.OP_Fwd_Run := NOT (NOT #Ctrl.OP_Fwd_Man AND NOT #Ctrl.OP_Fwd_Aut);
   #Ctrl.OP_Bwd_Run := NOT (NOT #Ctrl.OP_Bwd_Man AND NOT #Ctrl.OP_Bwd_Aut);
END_REGION

REGION Network 11: <+>
END_REGION

REGION Network 12: Condizioni movimento Operazione a Lavoro / Riposo
   RUNG wire#powerrail
      Contact( #CIn.Manager.Ax_1.Control_ON )
      Contact( #CIn.Manager.Ax_1.Bwd )
      wire#w1
      Coil( #Sts.OP_Bwd_Cnd )
   END_RUNG
   RUNG wire#powerrail
      Contact( #CIn.Manager.Ax_2.Control_ON )
      Contact( #CIn.Manager.Ax_2.Bwd )
   END_RUNG wire#w1
   RUNG wire#powerrail
      Contact( #AreaInterface.Man )
      I_Contact( #CIn.Manager.Ax_1.Control_ON )
      I_Contact( #CIn.Manager.Ax_2.Control_ON )
      Contact( #Sts.OP_CanMoveFreely )
   END_RUNG wire#w1
   RUNG wire#powerrail
      Contact( #CIn.Manager.Ax_1.Control_ON )
      Contact( #CIn.Manager.Ax_1.Fwd )
      wire#w2
      Coil( #Sts.OP_Fwd_Cnd )
   END_RUNG
   RUNG wire#powerrail
      Contact( #CIn.Manager.Ax_2.Control_ON )
      Contact( #CIn.Manager.Ax_2.Fwd )
   END_RUNG wire#w2
   RUNG wire#powerrail
      Contact( #AreaInterface.Man )
      I_Contact( #CIn.Manager.Ax_1.Control_ON )
      I_Contact( #CIn.Manager.Ax_2.Control_ON )
      Contact( #Sts.OP_CanMoveFreely )
   END_RUNG wire#w2
   // the same network as SCL:
   #Sts.OP_Bwd_Cnd := (#CIn.Manager.Ax_1.Control_ON AND #CIn.Manager.Ax_1.Bwd) OR (#CIn.Manager.Ax_2.Control_ON AND #CIn.Manager.Ax_2.Bwd) OR (#AreaInterface.Man AND NOT #CIn.Manager.Ax_1.Control_ON AND NOT #CIn.Manager.Ax_2.Control_ON AND #Sts.OP_CanMoveFreely);
   #Sts.OP_Fwd_Cnd := (#CIn.Manager.Ax_1.Control_ON AND #CIn.Manager.Ax_1.Fwd) OR (#CIn.Manager.Ax_2.Control_ON AND #CIn.Manager.Ax_2.Fwd) OR (#AreaInterface.Man AND NOT #CIn.Manager.Ax_1.Control_ON AND NOT #CIn.Manager.Ax_2.Control_ON AND #Sts.OP_CanMoveFreely);
END_REGION

REGION Network 13 (SCL): [Ax_1 + Ax_2] - CIn Manger
   // TRASFERIMENTO CIn MANAGER ALLA MACCHINA
   #Ax_1.CIn.Manager := #CIn.Manager.Ax_1;
   #Ax_2.CIn.Manager := #CIn.Manager.Ax_2;
END_REGION

REGION Network 14 (SCL): [Ax_1 + Ax_2] - Cin Manager Comando arresto / lavoro
   //
   #Ax_1.CIn.Manager.Bwd := #Ax_2.CIn.Manager.Bwd := FALSE;
   //************************************
   #Ax_1.CIn.Manager.Fwd := #Ax_2.CIn.Manager.Fwd := FALSE;
   //
   // CIn Manager  Control ON se ho un richiesta di comando attiva
   #Ax_1.CIn.Manager.Control_ON := #Ax_2.CIn.Manager.Control_ON := #Ctrl.OP_Fwd_Run OR #Ctrl.OP_Bwd_Run;

   // CIn Manager Brw se ho un richiesta di comando indietro attiva
   #Ax_1.CIn.Manager.Bwd := #Ax_2.CIn.Manager.Bwd := #Ctrl.OP_Bwd_Run AND #Sts.OP_Bwd_Cnd;

   // CIn Manager Frw se ho un richiesta di comando avanti attiva
   // Se la battuta di coda è alta attivo tutte e 2 le rulliere
   IF #Ctrl.OP_Fwd_Run AND #Sts.OP_Fwd_Cnd AND #CIn.CarroPareggCoda.BattutaVerticale.Rest THEN
       #Ax_1.CIn.Manager.Fwd := #Ax_2.CIn.Manager.Fwd := TRUE;


       // Se la battuta di coda è bassa attivo la rulliera 1 e la 2 rimane ferma
   ELSIF (#Ctrl.OP_Fwd_Run AND #Sts.OP_Fwd_Cnd) AND #CIn.CarroPareggCoda.BattutaVerticale.Work THEN
       #Ax_1.CIn.Manager.Fwd := TRUE;
       #Ax_2.CIn.Manager.Fwd := FALSE;
   END_IF;
END_REGION

REGION Network 15 (SCL): [Ax_1 + 2] - CIn Abilitazioni Stop Manager
   // CIn Manager Stop per richiesta apertura safety
   // 
   #Ax_1.CIn.Manager.EnableStopDoorOpeningReq := #CIn.Manager.Ax_1.EnableStopDoorOpeningReq;
   #Ax_2.CIn.Manager.EnableStopDoorOpeningReq := #CIn.Manager.Ax_2.EnableStopDoorOpeningReq;

   // CIn Manager Stop in fase delle macchine precedenti
   // 
   #Ax_1.CIn.Manager.EnableStopInPhase := #CIn.Manager.Ax_1.EnableStopInPhase;
   #Ax_2.CIn.Manager.EnableStopInPhase := #CIn.Manager.Ax_2.EnableStopInPhase;

   // CIn Manager Stop programmato configurabile a piacere
   // 
   #Ax_1.CIn.Manager.EnableStopProgrammed := #CIn.Manager.Ax_1.EnableStopProgrammed;
   #Ax_2.CIn.Manager.EnableStopProgrammed := #CIn.Manager.Ax_2.EnableStopProgrammed;
END_REGION

REGION Network 16: <+>
END_REGION

REGION Network 17: Warning manacanza condizioni esecuzione Operazione RIPOSO / LAVORO
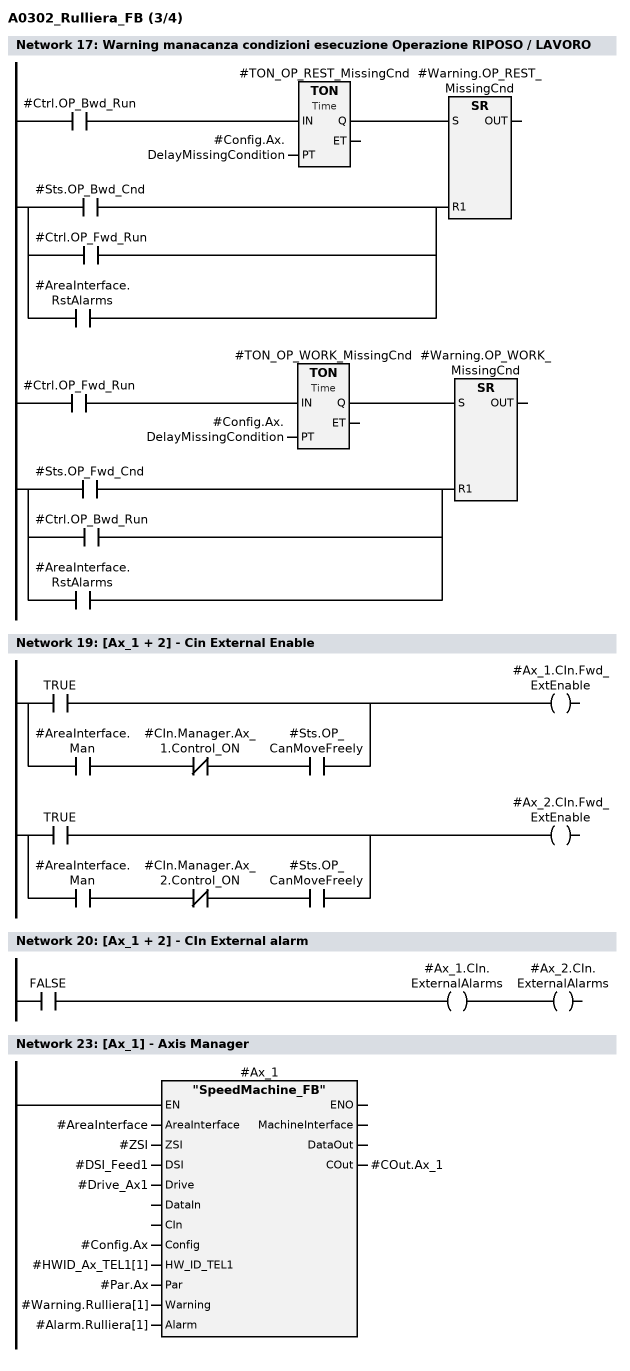
   RUNG wire#powerrail
      Contact( #Ctrl.OP_Bwd_Run )
      { S7_Templates := "time_type := Time" } #TON_OP_REST_MissingCnd.TON(pt := #Config.Ax.DelayMissingCondition, et =>)
      S_SR(operand := #Warning.OP_REST_MissingCnd, r1 := wire#w1)
   END_RUNG
   RUNG wire#powerrail
      Contact( #Sts.OP_Bwd_Cnd )
   END_RUNG wire#w1
   RUNG wire#powerrail
      Contact( #Ctrl.OP_Fwd_Run )
   END_RUNG wire#w1
   RUNG wire#powerrail
      Contact( #AreaInterface.RstAlarms )
   END_RUNG wire#w1
   RUNG wire#powerrail
      Contact( #Ctrl.OP_Fwd_Run )
      { S7_Templates := "time_type := Time" } #TON_OP_WORK_MissingCnd.TON(pt := #Config.Ax.DelayMissingCondition, et =>)
      S_SR(operand := #Warning.OP_WORK_MissingCnd, r1 := wire#w2)
   END_RUNG
   RUNG wire#powerrail
      Contact( #Sts.OP_Fwd_Cnd )
   END_RUNG wire#w2
   RUNG wire#powerrail
      Contact( #Ctrl.OP_Bwd_Run )
   END_RUNG wire#w2
   RUNG wire#powerrail
      Contact( #AreaInterface.RstAlarms )
   END_RUNG wire#w2
   // the same network as SCL:
   #TON_OP_REST_MissingCnd(IN := #Ctrl.OP_Bwd_Run, PT := #Config.Ax.DelayMissingCondition);   // TON
   IF #TON_OP_REST_MissingCnd.Q THEN
       #Warning.OP_REST_MissingCnd := TRUE;   // SR flip-flop
   END_IF;
   IF #Sts.OP_Bwd_Cnd OR #Ctrl.OP_Fwd_Run OR #AreaInterface.RstAlarms THEN
       #Warning.OP_REST_MissingCnd := FALSE;
   END_IF;
   #TON_OP_WORK_MissingCnd(IN := #Ctrl.OP_Fwd_Run, PT := #Config.Ax.DelayMissingCondition);   // TON
   IF #TON_OP_WORK_MissingCnd.Q THEN
       #Warning.OP_WORK_MissingCnd := TRUE;   // SR flip-flop
   END_IF;
   IF #Sts.OP_Fwd_Cnd OR #Ctrl.OP_Bwd_Run OR #AreaInterface.RstAlarms THEN
       #Warning.OP_WORK_MissingCnd := FALSE;
   END_IF;
END_REGION

REGION Network 18: <+>
END_REGION

REGION Network 19: [Ax_1 + 2] - Cin External Enable
   RUNG wire#powerrail
      Contact( TRUE )
      wire#w1
      Coil( #Ax_1.CIn.Fwd_ExtEnable )
   END_RUNG
   RUNG wire#powerrail
      Contact( #AreaInterface.Man )
      I_Contact( #CIn.Manager.Ax_1.Control_ON )
      Contact( #Sts.OP_CanMoveFreely )
   END_RUNG wire#w1
   RUNG wire#powerrail
      Contact( TRUE )
      wire#w2
      Coil( #Ax_2.CIn.Fwd_ExtEnable )
   END_RUNG
   RUNG wire#powerrail
      Contact( #AreaInterface.Man )
      I_Contact( #CIn.Manager.Ax_2.Control_ON )
      Contact( #Sts.OP_CanMoveFreely )
   END_RUNG wire#w2
   // the same network as SCL:
   #Ax_1.CIn.Fwd_ExtEnable := TRUE OR (#AreaInterface.Man AND NOT #CIn.Manager.Ax_1.Control_ON AND #Sts.OP_CanMoveFreely);
   #Ax_2.CIn.Fwd_ExtEnable := TRUE OR (#AreaInterface.Man AND NOT #CIn.Manager.Ax_2.Control_ON AND #Sts.OP_CanMoveFreely);
END_REGION

REGION Network 20: [Ax_1 + 2] - CIn External alarm
   RUNG wire#powerrail
      Contact( FALSE )
      Coil( #Ax_1.CIn.ExternalAlarms )
      Coil( #Ax_2.CIn.ExternalAlarms )
   END_RUNG
   // the same network as SCL:
   #Ax_1.CIn.ExternalAlarms := FALSE;
   #Ax_2.CIn.ExternalAlarms := FALSE;
END_REGION

REGION Network 21: <+>
END_REGION

REGION Network 22: <<< RULLIERA 1 >>>
END_REGION

REGION Network 23: [Ax_1] - Axis Manager
   RUNG wire#powerrail
      #Ax_1(AreaInterface := #AreaInterface, ZSI := #ZSI, DSI := #DSI_Feed1, Drive := #Drive_Ax1, DataIn :=, CIn :=, Config := #Config.Ax, HW_ID_TEL1 := #HWID_Ax_TEL1[1], Par := #Par.Ax, Warning := #Warning.Rulliera[1], Alarm := #Alarm.Rulliera[1], MachineInterface =>, DataOut =>, COut => #COut.Ax_1)
   END_RUNG
   // the same network as SCL:
   #Ax_1(AreaInterface := #AreaInterface,   // "SpeedMachine_FB"
         ZSI := #ZSI,
         DSI := #DSI_Feed1,
         Drive := #Drive_Ax1,
         Config := #Config.Ax,
         HW_ID_TEL1 := #HWID_Ax_TEL1[1],
         Par := #Par.Ax,
         Warning := #Warning.Rulliera[1],
         Alarm := #Alarm.Rulliera[1],
         COut => #COut.Ax_1);
END_REGION

REGION Network 24: <<< RULLIERA 2 >>>
END_REGION

REGION Network 25: [Ax_2] - Axis Manager
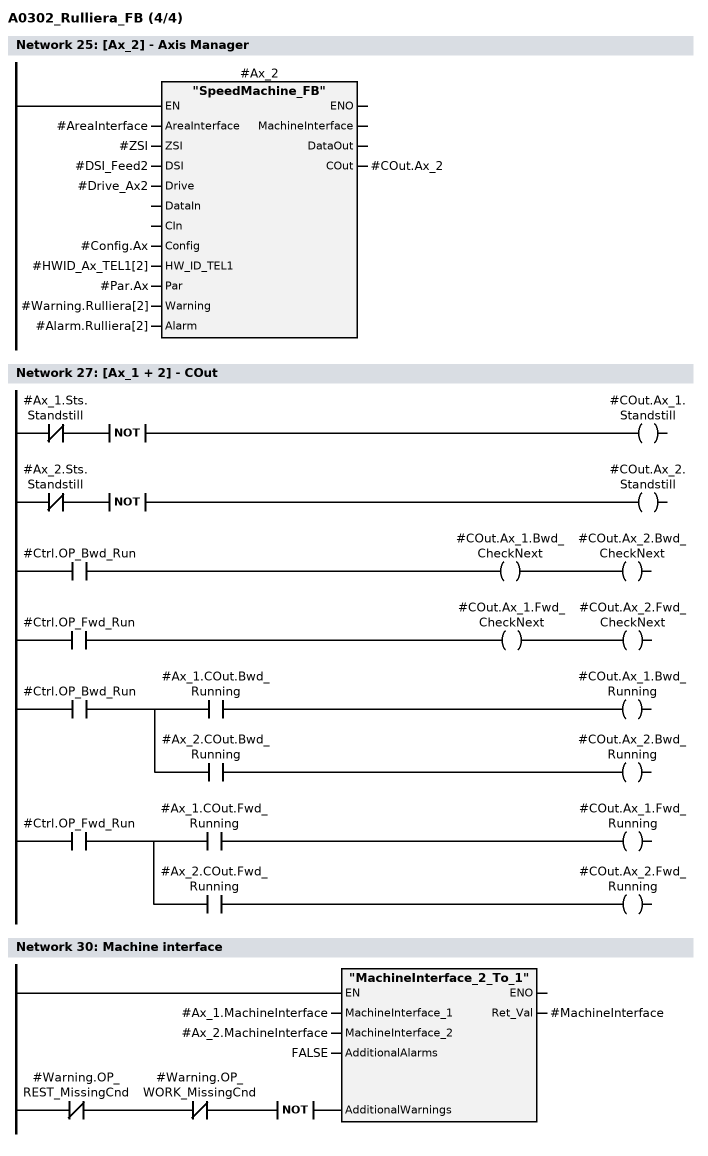
   RUNG wire#powerrail
      #Ax_2(AreaInterface := #AreaInterface, ZSI := #ZSI, DSI := #DSI_Feed2, Drive := #Drive_Ax2, DataIn :=, CIn :=, Config := #Config.Ax, HW_ID_TEL1 := #HWID_Ax_TEL1[2], Par := #Par.Ax, Warning := #Warning.Rulliera[2], Alarm := #Alarm.Rulliera[2], MachineInterface =>, DataOut =>, COut => #COut.Ax_2)
   END_RUNG
   // the same network as SCL:
   #Ax_2(AreaInterface := #AreaInterface,   // "SpeedMachine_FB"
         ZSI := #ZSI,
         DSI := #DSI_Feed2,
         Drive := #Drive_Ax2,
         Config := #Config.Ax,
         HW_ID_TEL1 := #HWID_Ax_TEL1[2],
         Par := #Par.Ax,
         Warning := #Warning.Rulliera[2],
         Alarm := #Alarm.Rulliera[2],
         COut => #COut.Ax_2);
END_REGION

REGION Network 27: [Ax_1 + 2] - COut
   RUNG wire#powerrail
      I_Contact( #Ax_1.Sts.Standstill )
      Not()
      Coil( #COut.Ax_1.Standstill )
   END_RUNG
   RUNG wire#powerrail
      I_Contact( #Ax_2.Sts.Standstill )
      Not()
      Coil( #COut.Ax_2.Standstill )
   END_RUNG
   RUNG wire#powerrail
      Contact( #Ctrl.OP_Bwd_Run )
      Coil( #COut.Ax_1.Bwd_CheckNext )
      Coil( #COut.Ax_2.Bwd_CheckNext )
   END_RUNG
   RUNG wire#powerrail
      Contact( #Ctrl.OP_Fwd_Run )
      Coil( #COut.Ax_1.Fwd_CheckNext )
      Coil( #COut.Ax_2.Fwd_CheckNext )
   END_RUNG
   RUNG wire#powerrail
      Contact( #Ctrl.OP_Bwd_Run )
      wire#w1
      Contact( #Ax_1.COut.Bwd_Running )
      Coil( #COut.Ax_1.Bwd_Running )
   END_RUNG
   RUNG wire#w1
      Contact( #Ax_2.COut.Bwd_Running )
      Coil( #COut.Ax_2.Bwd_Running )
   END_RUNG
   RUNG wire#powerrail
      Contact( #Ctrl.OP_Fwd_Run )
      wire#w2
      Contact( #Ax_1.COut.Fwd_Running )
      Coil( #COut.Ax_1.Fwd_Running )
   END_RUNG
   RUNG wire#w2
      Contact( #Ax_2.COut.Fwd_Running )
      Coil( #COut.Ax_2.Fwd_Running )
   END_RUNG
   // the same network as SCL:
   #COut.Ax_1.Standstill := NOT (NOT #Ax_1.Sts.Standstill);
   #COut.Ax_2.Standstill := NOT (NOT #Ax_2.Sts.Standstill);
   #COut.Ax_1.Bwd_CheckNext := #Ctrl.OP_Bwd_Run;
   #COut.Ax_2.Bwd_CheckNext := #Ctrl.OP_Bwd_Run;
   #COut.Ax_1.Fwd_CheckNext := #Ctrl.OP_Fwd_Run;
   #COut.Ax_2.Fwd_CheckNext := #Ctrl.OP_Fwd_Run;
   #COut.Ax_1.Bwd_Running := #Ctrl.OP_Bwd_Run AND #Ax_1.COut.Bwd_Running;
   #COut.Ax_2.Bwd_Running := #Ctrl.OP_Bwd_Run AND #Ax_2.COut.Bwd_Running;
   #COut.Ax_1.Fwd_Running := #Ctrl.OP_Fwd_Run AND #Ax_1.COut.Fwd_Running;
   #COut.Ax_2.Fwd_Running := #Ctrl.OP_Fwd_Run AND #Ax_2.COut.Fwd_Running;
END_REGION

REGION Network 29: <<< MACHINE STATUS >>>
END_REGION

REGION Network 30: Machine interface
   RUNG wire#powerrail
      "MachineInterface_2_To_1"(AdditionalWarnings := wire#w1, MachineInterface_1 := #Ax_1.MachineInterface, MachineInterface_2 := #Ax_2.MachineInterface, AdditionalAlarms := FALSE, Ret_Val => #MachineInterface)
   END_RUNG
   RUNG wire#powerrail
      I_Contact( #Warning.OP_REST_MissingCnd )
      I_Contact( #Warning.OP_WORK_MissingCnd )
      Not()
   END_RUNG wire#w1
   // the same network as SCL:
   #MachineInterface := "MachineInterface_2_To_1"(MachineInterface_1 := #Ax_1.MachineInterface,
                           MachineInterface_2 := #Ax_2.MachineInterface,
                           AdditionalAlarms := FALSE,
                           AdditionalWarnings := NOT (NOT #Warning.OP_REST_MissingCnd AND NOT #Warning.OP_WORK_MissingCnd));
END_REGION
END_FUNCTION_BLOCK

FUNCTION "A0302_Centratori_CALL" : Void   // FC97, LAD
// stored: SetENOAutomatically false
   VAR_TEMP
      Missing_Input : Bool;
      Missing_Output : Bool;
   END_VAR
BEGIN

REGION Network 1 (SCL): << TRASFERIMENTO stati CIn del blocco >>
   // SOSTITUIRE SYS BYPASS CON INGRESSI DIGITALI
   // TRASFERIMENTO COMANDI CIn MANAGER
   "A0302_Centratori".CIn.Manager := "A0302_Manager".COut.Rulliera.Centratori;
   //
   "A0302_Centratori".CIn.SemiAut_Pb := "A0302_Manager".DataIn.SemiAut_Pb;


   REGION TRASFERIMENTO STATI SENSORI RULLIERA 

       "A0302_Centratori".CIn.Rulliera.Coda.Sens.FTC_Rall := "A0302_Rulliera".IEC_FTC_CodaRall.FTC_On;
       "A0302_Centratori".CIn.Rulliera.Coda.Sens.FTC_Prox_Ing := "A0302_Rulliera".IEC_FTC_CodaProxIng.FTC_On;
       "A0302_Centratori".CIn.Rulliera.Centro.Sens.FTC_Centrale := "A0302_Rulliera".IEC_FTC_Centro.FTC_On;

   END_REGION ;

   REGION TRASFERIMENTO STATI CARRO PAREGGIATORE DI CODA

       "A0302_Centratori".CIn.CarroPareggCoda.Ax := "A0302_PareggiatoreCoda".COut.Ax;
       "A0302_Centratori".CIn.CarroPareggCoda.Bloccaggio := "A0302_PareggiatoreCoda".COut.Bloccaggio;
       "A0302_Centratori".CIn.CarroPareggCoda.BattutaVerticale := "A0302_PareggiatoreCoda".COut.BattutaVerticale;
       "A0302_Centratori".CIn.CarroPareggCoda.PareggiatoreLong := "A0302_PareggiatoreCoda".COut.PareggiatoreLong;
       "A0302_Centratori".CIn.CarroPareggCoda.Sens.FTC_Ingombro_In := "A0302_PareggiatoreCoda".IEC_FTC_Input.FTC_On;
       "A0302_Centratori".CIn.CarroPareggCoda.Sens.FTC_Ingombro_Out := "A0302_PareggiatoreCoda".IEC_FTC_Output.FTC_On;
       "A0302_Centratori".CIn.CarroPareggCoda.Sens.PresenzaMat := "A0302_PareggiatoreCoda".IEC_FTC_PresentMat.FTC_On;

   END_REGION ;

   REGION TRASFERIMENTO STATI CARRO PAREGGIATORE DI TESTA

       "A0302_Centratori".CIn.CarroPareggTesta.Ax := "A0302_PareggiatoreTesta".COut.Ax;
       "A0302_Centratori".CIn.CarroPareggTesta.Bloccaggio := "A0302_PareggiatoreTesta".COut.Bloccaggio;
       "A0302_Centratori".CIn.CarroPareggTesta.Centraggio := "A0302_PareggiatoreTesta".COut.Centraggio;
       "A0302_Centratori".CIn.CarroPareggTesta.Sollevatore := "A0302_PareggiatoreTesta".COut.Sollevatore;
       "A0302_Centratori".CIn.CarroPareggTesta.Sens.FTC1_Rall := "A0302_PareggiatoreTesta".IEC_FTC_Rall.FTC_On;
       "A0302_Centratori".CIn.CarroPareggTesta.Sens.FTC2_Prox_Ls := "A0302_PareggiatoreTesta".IEC_FTC_ProxLs.FTC_On;
       "A0302_Centratori".CIn.CarroPareggTesta.Sens.PresenzaMat := "A0302_PareggiatoreTesta".IEC_FTC_PresentMat.FTC_On;

   END_REGION ;

   // TRASFERIMENTO STATO DELLE ZONE INGRESSO E USCITA DELLA STAZIONE
   "A0302_Centratori".CIn.BTrk.ZoneA0302Entry_Empty := "A0302_Manager".Sts.BTrk.ZoneA0302Entry_Empty;
   "A0302_Centratori".CIn.BTrk.ZoneA0302Exit_Empty := "A0302_Manager".Sts.BTrk.ZoneA0302Exit_Empty;
END_REGION

REGION Network 2: <<< DATA IN >>>
END_REGION

REGION Network 3 (SCL): DATA In - Pulsanti OP
   // Pulsanti OP lavoro
   // 
   "A0302_Centratori".DataIn.OP.Rest := "A03_HMI".MB3.Button.A0302.Centratori.OP.Rest;
   "A0302_Centratori".DataIn.OP.Work := "A03_HMI".MB3.Button.A0302.Centratori.OP.Work;
END_REGION

REGION Network 4: DataIn - Centraggio 1
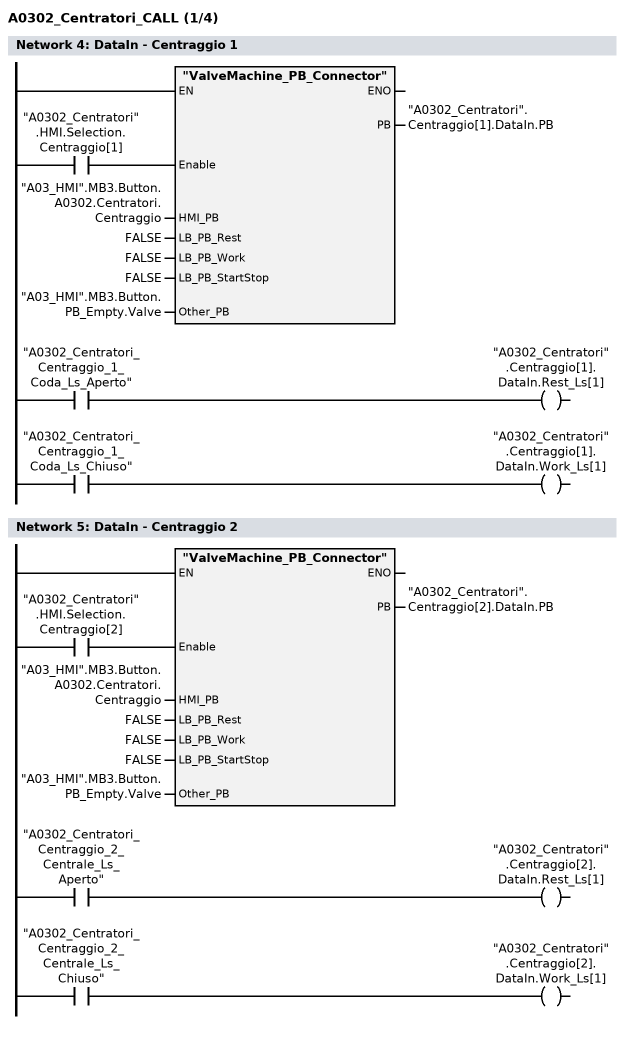
   RUNG wire#powerrail
      "ValveMachine_PB_Connector"(Enable := wire#w1, HMI_PB := "A03_HMI".MB3.Button.A0302.Centratori.Centraggio, LB_PB_Rest := FALSE, LB_PB_Work := FALSE, LB_PB_StartStop := FALSE, Other_PB := "A03_HMI".MB3.Button.PB_Empty.Valve, PB => "A0302_Centratori".Centraggio[1].DataIn.PB)
   END_RUNG
   RUNG wire#powerrail
      Contact( "A0302_Centratori".HMI.Selection.Centraggio[1] )
   END_RUNG wire#w1
   RUNG wire#powerrail
      Contact( "A0302_Centratori_Centraggio_1_Coda_Ls_Aperto" )
      Coil( "A0302_Centratori".Centraggio[1].DataIn.Rest_Ls[1] )
   END_RUNG
   RUNG wire#powerrail
      Contact( "A0302_Centratori_Centraggio_1_Coda_Ls_Chiuso" )
      Coil( "A0302_Centratori".Centraggio[1].DataIn.Work_Ls[1] )
   END_RUNG
   // the same network as SCL:
   "ValveMachine_PB_Connector"(Enable := "A0302_Centratori".HMI.Selection.Centraggio[1],
                           HMI_PB := "A03_HMI".MB3.Button.A0302.Centratori.Centraggio,
                           LB_PB_Rest := FALSE,
                           LB_PB_Work := FALSE,
                           LB_PB_StartStop := FALSE,
                           Other_PB := "A03_HMI".MB3.Button.PB_Empty.Valve,
                           PB => "A0302_Centratori".Centraggio[1].DataIn.PB);
   "A0302_Centratori".Centraggio[1].DataIn.Rest_Ls[1] := "A0302_Centratori_Centraggio_1_Coda_Ls_Aperto";
   "A0302_Centratori".Centraggio[1].DataIn.Work_Ls[1] := "A0302_Centratori_Centraggio_1_Coda_Ls_Chiuso";
END_REGION

REGION Network 5: DataIn - Centraggio 2
   RUNG wire#powerrail
      "ValveMachine_PB_Connector"(Enable := wire#w1, HMI_PB := "A03_HMI".MB3.Button.A0302.Centratori.Centraggio, LB_PB_Rest := FALSE, LB_PB_Work := FALSE, LB_PB_StartStop := FALSE, Other_PB := "A03_HMI".MB3.Button.PB_Empty.Valve, PB => "A0302_Centratori".Centraggio[2].DataIn.PB)
   END_RUNG
   RUNG wire#powerrail
      Contact( "A0302_Centratori".HMI.Selection.Centraggio[2] )
   END_RUNG wire#w1
   RUNG wire#powerrail
      Contact( "A0302_Centratori_Centraggio_2_Centrale_Ls_Aperto" )
      Coil( "A0302_Centratori".Centraggio[2].DataIn.Rest_Ls[1] )
   END_RUNG
   RUNG wire#powerrail
      Contact( "A0302_Centratori_Centraggio_2_Centrale_Ls_Chiuso" )
      Coil( "A0302_Centratori".Centraggio[2].DataIn.Work_Ls[1] )
   END_RUNG
   // the same network as SCL:
   "ValveMachine_PB_Connector"(Enable := "A0302_Centratori".HMI.Selection.Centraggio[2],
                           HMI_PB := "A03_HMI".MB3.Button.A0302.Centratori.Centraggio,
                           LB_PB_Rest := FALSE,
                           LB_PB_Work := FALSE,
                           LB_PB_StartStop := FALSE,
                           Other_PB := "A03_HMI".MB3.Button.PB_Empty.Valve,
                           PB => "A0302_Centratori".Centraggio[2].DataIn.PB);
   "A0302_Centratori".Centraggio[2].DataIn.Rest_Ls[1] := "A0302_Centratori_Centraggio_2_Centrale_Ls_Aperto";
   "A0302_Centratori".Centraggio[2].DataIn.Work_Ls[1] := "A0302_Centratori_Centraggio_2_Centrale_Ls_Chiuso";
END_REGION

REGION Network 6: DataIn - Centraggio 3
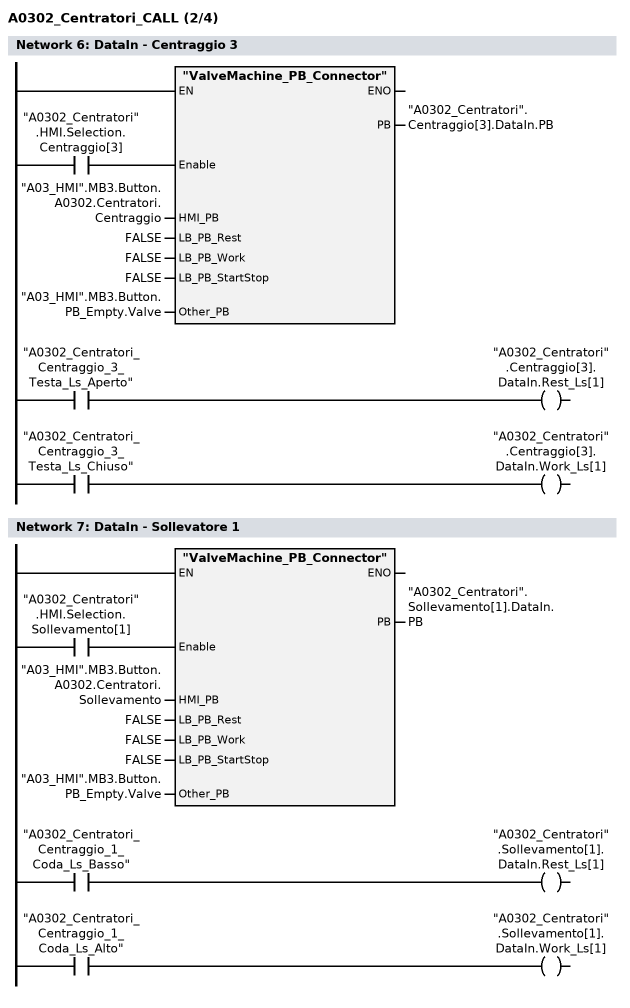
   RUNG wire#powerrail
      "ValveMachine_PB_Connector"(Enable := wire#w1, HMI_PB := "A03_HMI".MB3.Button.A0302.Centratori.Centraggio, LB_PB_Rest := FALSE, LB_PB_Work := FALSE, LB_PB_StartStop := FALSE, Other_PB := "A03_HMI".MB3.Button.PB_Empty.Valve, PB => "A0302_Centratori".Centraggio[3].DataIn.PB)
   END_RUNG
   RUNG wire#powerrail
      Contact( "A0302_Centratori".HMI.Selection.Centraggio[3] )
   END_RUNG wire#w1
   RUNG wire#powerrail
      Contact( "A0302_Centratori_Centraggio_3_Testa_Ls_Aperto" )
      Coil( "A0302_Centratori".Centraggio[3].DataIn.Rest_Ls[1] )
   END_RUNG
   RUNG wire#powerrail
      Contact( "A0302_Centratori_Centraggio_3_Testa_Ls_Chiuso" )
      Coil( "A0302_Centratori".Centraggio[3].DataIn.Work_Ls[1] )
   END_RUNG
   // the same network as SCL:
   "ValveMachine_PB_Connector"(Enable := "A0302_Centratori".HMI.Selection.Centraggio[3],
                           HMI_PB := "A03_HMI".MB3.Button.A0302.Centratori.Centraggio,
                           LB_PB_Rest := FALSE,
                           LB_PB_Work := FALSE,
                           LB_PB_StartStop := FALSE,
                           Other_PB := "A03_HMI".MB3.Button.PB_Empty.Valve,
                           PB => "A0302_Centratori".Centraggio[3].DataIn.PB);
   "A0302_Centratori".Centraggio[3].DataIn.Rest_Ls[1] := "A0302_Centratori_Centraggio_3_Testa_Ls_Aperto";
   "A0302_Centratori".Centraggio[3].DataIn.Work_Ls[1] := "A0302_Centratori_Centraggio_3_Testa_Ls_Chiuso";
END_REGION

REGION Network 7: DataIn - Sollevatore 1
   RUNG wire#powerrail
      "ValveMachine_PB_Connector"(Enable := wire#w1, HMI_PB := "A03_HMI".MB3.Button.A0302.Centratori.Sollevamento, LB_PB_Rest := FALSE, LB_PB_Work := FALSE, LB_PB_StartStop := FALSE, Other_PB := "A03_HMI".MB3.Button.PB_Empty.Valve, PB => "A0302_Centratori".Sollevamento[1].DataIn.PB)
   END_RUNG
   RUNG wire#powerrail
      Contact( "A0302_Centratori".HMI.Selection.Sollevamento[1] )
   END_RUNG wire#w1
   RUNG wire#powerrail
      Contact( "A0302_Centratori_Centraggio_1_Coda_Ls_Basso" )
      Coil( "A0302_Centratori".Sollevamento[1].DataIn.Rest_Ls[1] )
   END_RUNG
   RUNG wire#powerrail
      Contact( "A0302_Centratori_Centraggio_1_Coda_Ls_Alto" )
      Coil( "A0302_Centratori".Sollevamento[1].DataIn.Work_Ls[1] )
   END_RUNG
   // the same network as SCL:
   "ValveMachine_PB_Connector"(Enable := "A0302_Centratori".HMI.Selection.Sollevamento[1],
                           HMI_PB := "A03_HMI".MB3.Button.A0302.Centratori.Sollevamento,
                           LB_PB_Rest := FALSE,
                           LB_PB_Work := FALSE,
                           LB_PB_StartStop := FALSE,
                           Other_PB := "A03_HMI".MB3.Button.PB_Empty.Valve,
                           PB => "A0302_Centratori".Sollevamento[1].DataIn.PB);
   "A0302_Centratori".Sollevamento[1].DataIn.Rest_Ls[1] := "A0302_Centratori_Centraggio_1_Coda_Ls_Basso";
   "A0302_Centratori".Sollevamento[1].DataIn.Work_Ls[1] := "A0302_Centratori_Centraggio_1_Coda_Ls_Alto";
END_REGION

REGION Network 8: DataIn - Sollevatore 2
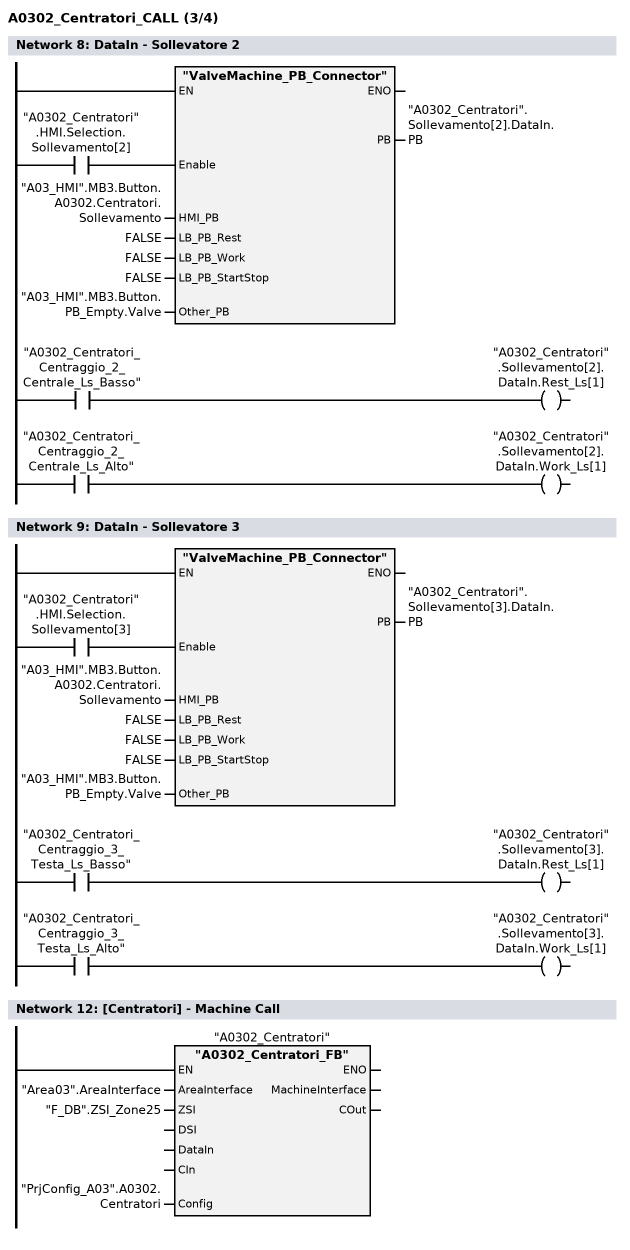
   RUNG wire#powerrail
      "ValveMachine_PB_Connector"(Enable := wire#w1, HMI_PB := "A03_HMI".MB3.Button.A0302.Centratori.Sollevamento, LB_PB_Rest := FALSE, LB_PB_Work := FALSE, LB_PB_StartStop := FALSE, Other_PB := "A03_HMI".MB3.Button.PB_Empty.Valve, PB => "A0302_Centratori".Sollevamento[2].DataIn.PB)
   END_RUNG
   RUNG wire#powerrail
      Contact( "A0302_Centratori".HMI.Selection.Sollevamento[2] )
   END_RUNG wire#w1
   RUNG wire#powerrail
      Contact( "A0302_Centratori_Centraggio_2_Centrale_Ls_Basso" )
      Coil( "A0302_Centratori".Sollevamento[2].DataIn.Rest_Ls[1] )
   END_RUNG
   RUNG wire#powerrail
      Contact( "A0302_Centratori_Centraggio_2_Centrale_Ls_Alto" )
      Coil( "A0302_Centratori".Sollevamento[2].DataIn.Work_Ls[1] )
   END_RUNG
   // the same network as SCL:
   "ValveMachine_PB_Connector"(Enable := "A0302_Centratori".HMI.Selection.Sollevamento[2],
                           HMI_PB := "A03_HMI".MB3.Button.A0302.Centratori.Sollevamento,
                           LB_PB_Rest := FALSE,
                           LB_PB_Work := FALSE,
                           LB_PB_StartStop := FALSE,
                           Other_PB := "A03_HMI".MB3.Button.PB_Empty.Valve,
                           PB => "A0302_Centratori".Sollevamento[2].DataIn.PB);
   "A0302_Centratori".Sollevamento[2].DataIn.Rest_Ls[1] := "A0302_Centratori_Centraggio_2_Centrale_Ls_Basso";
   "A0302_Centratori".Sollevamento[2].DataIn.Work_Ls[1] := "A0302_Centratori_Centraggio_2_Centrale_Ls_Alto";
END_REGION

